KUKA KRL program: MyProgram_080().src

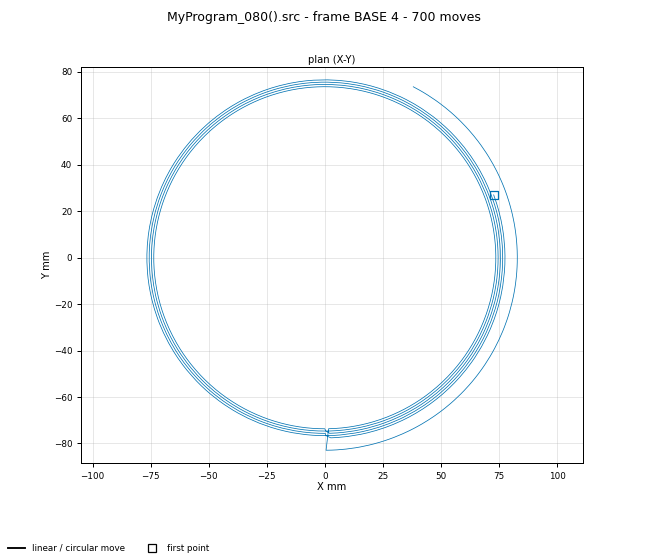
[picture p0: tool path of MyProgram_080().src in frame BASE 4, 700 of 700 moves have a stored position in this frame; points joined in program order, loops and branches not executed]
&ACCESS RVP
&REL 1
&PARAM TEMPLATE = C:\KRC\Roboter\Template\vorgabe
&PARAM EDITMASK = *
DEF MyProgram_080()
; ---- Setting reference (Base) ----
$BASE = BASE_DATA[4]

; --------------------------
; ---- Setting tool (TCP) ----
$TOOL = TOOL_DATA[3]
; --------------------------

$VEL.CP = VEL_APROX_PRINT
Startdeposition()
$VEL.CP = VEL_PRINT
LIN {X 72.7406,Y 27.0549,Z 81,A 13.4296,B 24.8995,C -2.3141,E1 25.1512,E2 431.179} C_DIS
LIN {X 74.0398,Y 23.263,Z 81,A 11.6779,B 24.8971,C -2.342,E1 25.1526,E2 432.855} C_DIS
LIN {X 75.0363,Y 19.8168,Z 81,A 8.2037,B 24.9,C -2.3088,E1 25.1553,E2 436.3875} C_DIS
LIN {X 75.8768,Y 16.3012,Z 81,A 6.032,B 24.8994,C -2.3158,E1 25.1566,E2 438.5303} C_DIS
LIN {X 76.4846,Y 13.161,Z 81,A 2.9896,B 24.9018,C -2.2877,E1 25.1581,E2 441.6211} C_DIS
LIN {X 77.0242,Y 9.5105,Z 81,A -0.3457,B 24.9041,C -2.2607,E1 25.1592,E2 445.0004} C_DIS
LIN {X 77.5014,Y 4.0671,Z 81,A -2.5659,B 24.9005,C -2.3033,E1 25.1596,E2 447.1069} C_DIS
LIN {X 77.6032,Y 0.8398,Z 81,A -5.5015,B 24.9026,C -2.2787,E1 25.1598,E2 450.0831} C_DIS
LIN {X 77.5585,Y -2.7704,Z 81,A -8.1214,B 24.9032,C -2.2716,E1 25.1596,E2 452.7042} C_DIS
LIN {X 77.3829,Y -5.9099,Z 81,A -10.3219,B 24.9035,C -2.2679,E1 25.1592,E2 454.9004} C_DIS
LIN {X 76.6451,Y -12.1903,Z 81,A -14.3809,B 24.9032,C -2.2718,E1 25.1578,E2 458.926} C_DIS
LIN {X 75.7643,Y -16.8174,Z 81,A -18.4569,B 24.9057,C -2.2423,E1 25.1557,E2 463.048} C_DIS
LIN {X 74.816,Y -20.6292,Z 81,A -21.3337,B 24.9064,C -2.2339,E1 25.1536,E2 465.928} C_DIS
LIN {X 74.0707,Y -23.163,Z 81,A -23.9313,B 24.9085,C -2.208,E1 25.1514,E2 468.5719} C_DIS
LIN {X 72.9129,Y -26.5834,Z 81,A -25.729,B 24.907,C -2.2264,E1 25.1498,E2 470.3162} C_DIS
LIN {X 71.3683,Y -30.4905,Z 81,A -29.3108,B 24.909,C -2.2023,E1 25.1459,E2 473.9352} C_DIS
LIN {X 69.9864,Y -33.5391,Z 81,A -31.3794,B 24.9086,C -2.2072,E1 25.1435,E2 475.981} C_DIS
LIN {X 67.4557,Y -38.3768,Z 81,A -35.2444,B 24.9092,C -2.2005,E1 25.1385,E2 479.8414} C_DIS
LIN {X 64.6383,Y -42.9527,Z 81,A -39.0995,B 24.9098,C -2.1927,E1 25.1328,E2 483.6954} C_DIS
LIN {X 63.2802,Y -44.929,Z 81,A -41.4223,B 24.9116,C -2.1711,E1 25.129,E2 486.0579} C_DIS
LIN {X 60.7597,Y -48.2832,Z 81,A -44.696,B 24.9127,C -2.1576,E1 25.1233,E2 489.3481} C_DIS
LIN {X 57.9727,Y -51.5963,Z 81,A -47.345,B 24.912,C -2.1659,E1 25.1185,E2 491.9656} C_DIS
LIN {X 55.8853,Y -53.8498,Z 81,A -50.1831,B 24.9139,C -2.1432,E1 25.113,E2 494.845} C_DIS
LIN {X 53.6172,Y -56.1095,Z 81,A -52.4693,B 24.9141,C -2.1399,E1 25.1084,E2 497.1295} C_DIS
LIN {X 50.5856,Y -58.8573,Z 81,A -55.0251,B 24.9136,C -2.1469,E1 25.1031,E2 499.6587} C_DIS
LIN {X 47.9048,Y -61.0588,Z 81,A -58.0995,B 24.9152,C -2.1261,E1 25.0963,E2 502.7707} C_DIS
LIN {X 45.3423,Y -62.9853,Z 81,A -59.9833,B 24.9145,C -2.1355,E1 25.0921,E2 504.6256} C_DIS
LIN {X 42.1438,Y -65.1685,Z 81,A -62.7724,B 24.9147,C -2.132,E1 25.0856,E2 507.4137} C_DIS
LIN {X 39.2698,Y -66.9396,Z 81,A -65.8722,B 24.9165,C -2.1096,E1 25.0781,E2 510.5569} C_DIS
LIN {X 36.2702,Y -68.6109,Z 81,A -67.2909,B 24.9143,C -2.138,E1 25.0748,E2 511.9043} C_DIS
LIN {X 33.3708,Y -70.0673,Z 81,A -69.9592,B 24.9152,C -2.1261,E1 25.068,E2 514.5937} C_DIS
LIN {X 29.4831,Y -71.7898,Z 81,A -73.2723,B 24.916,C -2.1164,E1 25.0595,E2 517.9219} C_DIS
LIN {X 26.0178,Y -73.117,Z 81,A -76.3261,B 24.917,C -2.1037,E1 25.0514,E2 520.9993} C_DIS
LIN {X 22.0037,Y -74.4232,Z 81,A -79.548,B 24.9175,C -2.0971,E1 25.0428,E2 524.2311} C_DIS
LIN {X 18.2814,Y -75.4238,Z 81,A -82.1856,B 24.9173,C -2.1002,E1 25.0357,E2 526.8574} C_DIS
LIN {X 15.4169,Y -76.0613,Z 81,A -84.1498,B 24.917,C -2.104,E1 25.0304,E2 528.8101} C_DIS
LIN {X 9.6899,Y -77.001,Z 81,A -88.5998,B 24.9176,C -2.0963,E1 25.0181,E2 533.2742} C_DIS
LIN {X 5.5154,Y -77.412,Z 81,A -91.4129,B 24.9171,C -2.1027,E1 25.0103,E2 536.0705} C_DIS
LIN {X 2.6067,Y -77.5643,Z 81,A -94.2953,B 24.9187,C -2.0816,E1 25.0021,E2 539.0022} C_DIS
LIN {X 2.6067,Y -77.5643,Z 81,A -94.2953,B 24.9187,C -2.0816,E1 25.0021,E2 539.0022} C_DIS
Enddeposition()
LIN {X 0.5051,Y -76.6088,Z 81,A -94.3061,B 24.914,C -2.1414,E1 25.0025,E2 538.871} C_DIS
Startdeposition()
$VEL.CP = VEL_PRINT
LIN {X 4.0039,Y -76.5168,Z 81,A -91.5176,B 24.9135,C -2.147,E1 25.0103,E2 536.0701} C_DIS
LIN {X 6.6768,Y -76.3306,Z 81,A -88.9313,B 24.9121,C -2.1645,E1 25.0176,E2 533.4436} C_DIS
LIN {X 13.1371,Y -75.4878,Z 81,A -84.5808,B 24.9131,C -2.1529,E1 25.0295,E2 529.1246} C_DIS
LIN {X 16.3512,Y -74.8562,Z 81,A -81.8311,B 24.9122,C -2.1637,E1 25.0371,E2 526.3527} C_DIS
LIN {X 19.7049,Y -74.0442,Z 81,A -79.2366,B 24.9119,C -2.1668,E1 25.0441,E2 523.755} C_DIS
LIN {X 23.4743,Y -72.9368,Z 81,A -76.6561,B 24.9125,C -2.1598,E1 25.0509,E2 521.1957} C_DIS
LIN {X 27.6858,Y -71.4453,Z 81,A -72.2914,B 24.9097,C -2.1944,E1 25.0625,E2 516.7584} C_DIS
LIN {X 31.9466,Y -69.6448,Z 81,A -69.902,B 24.9118,C -2.1679,E1 25.0684,E2 514.4377} C_DIS
LIN {X 33.9734,Y -68.6776,Z 81,A -67.9436,B 24.911,C -2.1789,E1 25.0734,E2 512.4585} C_DIS
LIN {X 38.7843,Y -66.0801,Z 81,A -64.0702,B 24.9109,C -2.1796,E1 25.0828,E2 508.5947} C_DIS
LIN {X 42.9281,Y -63.4664,Z 81,A -60.3035,B 24.9101,C -2.1898,E1 25.0917,E2 504.8164} C_DIS
LIN {X 45.9892,Y -61.2839,Z 81,A -57.4169,B 24.9094,C -2.1978,E1 25.0982,E2 501.921} C_DIS
LIN {X 49.171,Y -58.7629,Z 81,A -54.79,B 24.9099,C -2.1922,E1 25.1038,E2 499.3174} C_DIS
LIN {X 52.9625,Y -55.3703,Z 81,A -50.8405,B 24.9088,C -2.2053,E1 25.112,E2 495.3528} C_DIS
LIN {X 55.8207,Y -52.4867,Z 81,A -47.8961,B 24.9084,C -2.21,E1 25.1177,E2 492.4101} C_DIS
LIN {X 57.6696,Y -50.4483,Z 81,A -45.6064,B 24.9074,C -2.2222,E1 25.122,E2 490.1017} C_DIS
LIN {X 60.1141,Y -47.5089,Z 81,A -42.7917,B 24.9069,C -2.2284,E1 25.1269,E2 487.2855} C_DIS
LIN {X 63.1802,Y -43.3507,Z 81,A -39.3763,B 24.9071,C -2.2251,E1 25.1324,E2 483.8943} C_DIS
LIN {X 64.7091,Y -41.0307,Z 81,A -36.7547,B 24.9052,C -2.2476,E1 25.1365,E2 481.2326} C_DIS
LIN {X 66.493,Y -38.0722,Z 81,A -33.737,B 24.9035,C -2.2685,E1 25.1407,E2 478.1813} C_DIS
LIN {X 68.3146,Y -34.6981,Z 81,A -31.6623,B 24.9048,C -2.2523,E1 25.1433,E2 476.1557} C_DIS
LIN {X 69.6675,Y -31.8972,Z 81,A -29.3502,B 24.9043,C -2.2588,E1 25.1461,E2 473.8409} C_DIS
LIN {X 71.6458,Y -27.1604,Z 81,A -25.8048,B 24.9041,C -2.2614,E1 25.1498,E2 470.3089} C_DIS
LIN {X 73.3926,Y -22.0088,Z 81,A -20.8861,B 24.9007,C -2.3003,E1 25.1541,E2 465.326} C_DIS
LIN {X 74.2916,Y -18.7529,Z 81,A -18.9852,B 24.9017,C -2.2888,E1 25.1554,E2 463.4633} C_DIS
LIN {X 74.9344,Y -15.9924,Z 81,A -16.2071,B 24.8994,C -2.316,E1 25.157,E2 460.6372} C_DIS
LIN {X 75.589,Y -12.5348,Z 81,A -14.9013,B 24.9022,C -2.2833,E1 25.1576,E2 459.4164} C_DIS
LIN {X 76.1441,Y -8.5448,Z 81,A -11.2664,B 24.8997,C -2.312,E1 25.159,E2 455.735} C_DIS
LIN {X 76.4322,Y -5.3825,Z 81,A -8.9577,B 24.8992,C -2.3176,E1 25.1595,E2 453.4269} C_DIS
LIN {X 76.614,Y -1.0935,Z 81,A -5.0295,B 24.8964,C -2.3501,E1 25.1598,E2 449.4452} C_DIS
LIN {X 76.5801,Y 2.5132,Z 81,A -3.0751,B 24.8976,C -2.3356,E1 25.1596,E2 447.5368} C_DIS
LIN {X 76.4465,Y 5.1709,Z 81,A -0.1808,B 24.8946,C -2.37,E1 25.1591,E2 444.5783} C_DIS
LIN {X 76.0454,Y 9.3872,Z 81,A 2.5015,B 24.8951,C -2.3648,E1 25.1582,E2 441.9243} C_DIS
LIN {X 75.3914,Y 13.6729,Z 81,A 5.2733,B 24.8955,C -2.3603,E1 25.1569,E2 439.1792} C_DIS
LIN {X 74.78,Y 16.7004,Z 81,A 7.3071,B 24.8955,C -2.3589,E1 25.1558,E2 437.1606} C_DIS
LIN {X 74.058,Y 19.6555,Z 81,A 9.8384,B 24.8943,C -2.3737,E1 25.154,E2 434.609} C_DIS
LIN {X 73.1811,Y 22.7009,Z 81,A 12.5126,B 24.8928,C -2.3901,E1 25.1518,E2 431.9112} C_DIS
LIN {X 71.4621,Y 27.643,Z 81,A 16.0873,B 24.8928,C -2.3912,E1 25.1484,E2 428.354} C_DIS
LIN {X 70.1766,Y 30.7583,Z 81,A 19.1342,B 24.8906,C -2.4145,E1 25.145,E2 425.2688} C_DIS
LIN {X 68.8247,Y 33.6767,Z 81,A 21.4682,B 24.8902,C -2.4189,E1 25.1422,E2 422.9367} C_DIS
LIN {X 66.6712,Y 37.762,Z 81,A 24.2393,B 24.8912,C -2.4075,E1 25.1385,E2 420.2072} C_DIS
LIN {X 64.9518,Y 40.6456,Z 81,A 27.0598,B 24.8898,C -2.4234,E1 25.1344,E2 417.3634} C_DIS
LIN {X 62.8872,Y 43.7722,Z 81,A 30.8514,B 24.8864,C -2.4605,E1 25.1282,E2 413.5028} C_DIS
LIN {X 59.9348,Y 47.7358,Z 81,A 33.3959,B 24.8888,C -2.4344,E1 25.124,E2 411.0319} C_DIS
LIN {X 56.4841,Y 51.7721,Z 81,A 37.3342,B 24.888,C -2.4424,E1 25.1168,E2 407.0924} C_DIS
LIN {X 54.1841,Y 54.1766,Z 81,A 39.8561,B 24.8875,C -2.4487,E1 25.1118,E2 404.5664} C_DIS
LIN {X 51.7923,Y 56.4656,Z 81,A 42.128,B 24.8875,C -2.4477,E1 25.1072,E2 402.3062} C_DIS
LIN {X 48.7055,Y 59.1498,Z 81,A 45.1069,B 24.8872,C -2.4512,E1 25.1009,E2 399.3306} C_DIS
LIN {X 46.6152,Y 60.8101,Z 81,A 47.6684,B 24.8854,C -2.4714,E1 25.0952,E2 396.7308} C_DIS
LIN {X 41.6987,Y 64.2818,Z 81,A 51.863,B 24.8855,C -2.4697,E1 25.0855,E2 392.5543} C_DIS
LIN {X 38.5101,Y 66.2414,Z 81,A 54.7369,B 24.8849,C -2.476,E1 25.0786,E2 389.6745} C_DIS
LIN {X 35.0593,Y 68.13,Z 81,A 57.0933,B 24.8861,C -2.4631,E1 25.0729,E2 387.3554} C_DIS
LIN {X 32.717,Y 69.2862,Z 81,A 59.1876,B 24.8855,C -2.4695,E1 25.0676,E2 385.2515} C_DIS
LIN {X 27.6315,Y 71.4666,Z 81,A 64.03,B 24.8833,C -2.4938,E1 25.055,E2 380.3626} C_DIS
LIN {X 23.197,Y 73.0265,Z 81,A 67.0652,B 24.8843,C -2.4831,E1 25.0471,E2 377.3587} C_DIS
LIN {X 19.8161,Y 74.0146,Z 81,A 69.7453,B 24.884,C -2.4861,E1 25.0399,E2 374.6758} C_DIS
LIN {X 17.0226,Y 74.7067,Z 81,A 72.5334,B 24.8822,C -2.5051,E1 25.0322,E2 371.8465} C_DIS
LIN {X 13.6277,Y 75.3993,Z 81,A 74.4093,B 24.884,C -2.4862,E1 25.0272,E2 370.0177} C_DIS
LIN {X 10.5424,Y 75.8928,Z 81,A 76.8912,B 24.8835,C -2.4908,E1 25.0203,E2 367.527} C_DIS
LIN {X 5.9796,Y 76.3876,Z 81,A 80.7325,B 24.8825,C -2.5024,E1 25.0095,E2 363.6603} C_DIS
LIN {X 1.1387,Y 76.6132,Z 81,A 83.7746,B 24.884,C -2.4862,E1 25.0011,E2 360.6576} C_DIS
LIN {X -4.837,Y 76.4691,Z 81,A 88.3402,B 24.8839,C -2.4873,E1 24.9884,E2 356.0885} C_DIS
LIN {X -8.0265,Y 76.1996,Z 81,A 90.8059,B 24.8839,C -2.4881,E1 24.9815,E2 353.6197} C_DIS
LIN {X -11.1013,Y 75.8128,Z 81,A 93.1912,B 24.8838,C -2.4885,E1 24.9749,E2 351.2316} C_DIS
LIN {X -14.9837,Y 75.1429,Z 81,A 96.2499,B 24.8838,C -2.4891,E1 24.9665,E2 348.168} C_DIS
LIN {X -19.4527,Y 74.1117,Z 81,A 99.3472,B 24.8848,C -2.4771,E1 24.9582,E2 345.0951} C_DIS
LIN {X -22.985,Y 73.0928,Z 81,A 102.6998,B 24.8836,C -2.4899,E1 24.9491,E2 341.7062} C_DIS
LIN {X -26.3966,Y 71.9309,Z 81,A 105.7925,B 24.883,C -2.497,E1 24.941,E2 338.5905} C_DIS
LIN {X -30.2905,Y 70.3805,Z 81,A 107.9496,B 24.8858,C -2.467,E1 24.9356,E2 336.4998} C_DIS
LIN {X -34.5136,Y 68.4089,Z 81,A 111.2486,B 24.8867,C -2.4569,E1 24.9273,E2 333.2166} C_DIS
LIN {X -37.0817,Y 67.0511,Z 81,A 114.3662,B 24.8848,C -2.4775,E1 24.9195,E2 330.0411} C_DIS
LIN {X -40.0695,Y 65.3096,Z 81,A 116.3389,B 24.8867,C -2.457,E1 24.9149,E2 328.1109} C_DIS
LIN {X -42.8077,Y 63.5479,Z 81,A 118.7363,B 24.8872,C -2.4514,E1 24.9093,E2 325.719} C_DIS
LIN {X -46.5848,Y 60.8335,Z 81,A 122.3377,B 24.8876,C -2.4474,E1 24.9012,E2 322.1144} C_DIS
LIN {X -50.0446,Y 58.0221,Z 81,A 125.6479,B 24.8883,C -2.4395,E1 24.8941,E2 318.8104} C_DIS
LIN {X -53.7369,Y 54.6184,Z 81,A 129.1445,B 24.8897,C -2.4244,E1 24.8871,E2 315.3356} C_DIS
LIN {X -57.3893,Y 50.7688,Z 81,A 133.4156,B 24.8899,C -2.4221,E1 24.8789,E2 311.0512} C_DIS
LIN {X -60.4351,Y 47.1018,Z 81,A 136.9866,B 24.8907,C -2.413,E1 24.8726,E2 307.4854} C_DIS
LIN {X -63.3473,Y 43.104,Z 81,A 140.6648,B 24.8917,C -2.4025,E1 24.8667,E2 303.8143} C_DIS
LIN {X -65.1312,Y 40.3584,Z 81,A 142.8724,B 24.8928,C -2.3898,E1 24.8634,E2 301.6259} C_DIS
LIN {X -66.5326,Y 38.0034,Z 81,A 145.6655,B 24.8917,C -2.4021,E1 24.8594,E2 298.7886} C_DIS
LIN {X -68.4996,Y 34.3325,Z 81,A 148.3984,B 24.8934,C -2.3837,E1 24.856,E2 296.0852} C_DIS
LIN {X -70.2882,Y 30.5022,Z 81,A 152.0408,B 24.8932,C -2.3861,E1 24.8518,E2 292.4171} C_DIS
LIN {X -72.1333,Y 25.8416,Z 81,A 155.6738,B 24.8944,C -2.3718,E1 24.8483,E2 288.7978} C_DIS
LIN {X -73.6813,Y 21.0213,Z 81,A 158.6352,B 24.8972,C -2.3401,E1 24.8459,E2 285.895} C_DIS
LIN {X -74.47,Y 18.0288,Z 81,A 161.9607,B 24.8957,C -2.3573,E1 24.8436,E2 282.5089} C_DIS
LIN {X -75.456,Y 13.3139,Z 81,A 165.5401,B 24.8968,C -2.3454,E1 24.8417,E2 278.9368} C_DIS
LIN {X -75.994,Y 9.7835,Z 81,A 168.0798,B 24.8978,C -2.3337,E1 24.8408,E2 276.4099} C_DIS
LIN {X -76.4323,Y 5.3805,Z 81,A 171.932,B 24.8976,C -2.3365,E1 24.8399,E2 272.528} C_DIS
LIN {X -76.6084,Y 1.3996,Z 81,A 173.9908,B 24.9004,C -2.3045,E1 24.8398,E2 270.533} C_DIS
LIN {X -76.6007,Y -1.8197,Z 81,A 176.6959,B 24.9004,C -2.3041,E1 24.8398,E2 267.8127} C_DIS
LIN {X -76.3769,Y -6.1134,Z 81,A 179.7575,B 24.9016,C -2.2902,E1 24.8404,E2 264.7659} C_DIS
LIN {X -76.1095,Y -8.8402,Z 81,A -178.3528,B 24.9025,C -2.2799,E1 24.841,E2 262.8894} C_DIS
LIN {X -75.6777,Y -11.9906,Z 81,A -175.8658,B 24.9029,C -2.2752,E1 24.842,E2 260.399} C_DIS
LIN {X -75.009,Y -15.6367,Z 81,A -172.9725,B 24.9034,C -2.2696,E1 24.8436,E2 257.5019} C_DIS
LIN {X -74.4931,Y -17.9342,Z 81,A -170.2891,B 24.9019,C -2.2869,E1 24.8454,E2 254.7614} C_DIS
LIN {X -73.3805,Y -22.0494,Z 81,A -168.4859,B 24.9056,C -2.2434,E1 24.8467,E2 253.0518} C_DIS
LIN {X -72.0133,Y -26.1704,Z 81,A -164.7612,B 24.9054,C -2.2454,E1 24.8501,E2 249.3009} C_DIS
LIN {X -71.2631,Y -28.1496,Z 81,A -162.1753,B 24.9037,C -2.2658,E1 24.8528,E2 246.6519} C_DIS
LIN {X -69.5373,Y -32.1776,Z 81,A -159.9047,B 24.9066,C -2.2315,E1 24.8554,E2 244.4507} C_DIS
LIN {X -67.2711,Y -36.6801,Z 81,A -155.6898,B 24.9066,C -2.2323,E1 24.8608,E2 240.2115} C_DIS
LIN {X -65.0604,Y -40.4719,Z 81,A -152.7829,B 24.908,C -2.2144,E1 24.865,E2 237.3324} C_DIS
LIN {X -63.2183,Y -43.2936,Z 81,A -149.4449,B 24.9068,C -2.2287,E1 24.8703,E2 233.9437} C_DIS
LIN {X -60.9614,Y -46.4188,Z 81,A -147.5845,B 24.9096,C -2.1958,E1 24.8733,E2 232.1526} C_DIS
LIN {X -59.3245,Y -48.4924,Z 81,A -144.8184,B 24.9083,C -2.2112,E1 24.8782,E2 229.3369} C_DIS
LIN {X -55.4047,Y -52.9267,Z 81,A -140.8853,B 24.9101,C -2.1889,E1 24.8855,E2 225.4397} C_DIS
LIN {X -53.325,Y -55.0208,Z 81,A -138.8378,B 24.9108,C -2.1803,E1 24.8896,E2 223.4041} C_DIS
LIN {X -51.2072,Y -56.9969,Z 81,A -136.5265,B 24.9108,C -2.1797,E1 24.8944,E2 221.0849} C_DIS
LIN {X -49.3438,Y -58.6179,Z 81,A -134.3506,B 24.9105,C -2.1847,E1 24.899,E2 218.8886} C_DIS
LIN {X -45.6253,Y -61.555,Z 81,A -130.9776,B 24.9113,C -2.1741,E1 24.9065,E2 215.5287} C_DIS
LIN {X -43.143,Y -63.3209,Z 81,A -127.855,B 24.9098,C -2.1926,E1 24.9138,E2 212.3516} C_DIS
LIN {X -39.5137,Y -65.6474,Z 81,A -125.4562,B 24.912,C -2.166,E1 24.9194,E2 210.0085} C_DIS
LIN {X -37.3266,Y -66.9143,Z 81,A -123.4615,B 24.912,C -2.1662,E1 24.9243,E2 208.0076} C_DIS
LIN {X -33.0427,Y -69.1304,Z 81,A -119.5685,B 24.9117,C -2.1695,E1 24.9341,E2 204.0965} C_DIS
LIN {X -28.1562,Y -71.2605,Z 81,A -115.906,B 24.9128,C -2.1567,E1 24.9434,E2 200.4561} C_DIS
LIN {X -23.2066,Y -73.0234,Z 81,A -112.0862,B 24.9133,C -2.1506,E1 24.9535,E2 196.6437} C_DIS
LIN {X -20.0867,Y -73.9415,Z 81,A -108.9851,B 24.9119,C -2.1673,E1 24.962,E2 193.4979} C_DIS
LIN {X -16.5756,Y -74.8072,Z 81,A -107.0751,B 24.9138,C -2.1442,E1 24.967,E2 191.6403} C_DIS
LIN {X -13.7391,Y -75.3795,Z 81,A -104.6203,B 24.9132,C -2.1514,E1 24.9738,E2 189.1658} C_DIS
LIN {X -8.4181,Y -76.1586,Z 81,A -100.772,B 24.9136,C -2.1458,E1 24.9845,E2 185.3279} C_DIS
LIN {X -5.3144,Y -76.4368,Z 81,A -98.4403,B 24.9136,C -2.1458,E1 24.9909,E2 182.9952} C_DIS
LIN {X -2.5364,Y -76.5794,Z 81,A -96.1753,B 24.9132,C -2.1512,E1 24.9973,E2 180.7169} C_DIS
LIN {X 0.5051,Y -76.6088,Z 81,A -94.3042,B 24.9141,C -2.1406,E1 25.0025,E2 178.871} C_DIS
Enddeposition()
LIN {X 0.5051,Y -76.6088,Z 81,A -94.3042,B 24.9141,C -2.1406,E1 25.0025,E2 178.871} C_DIS
Startdeposition()
$VEL.CP = VEL_PRINT
LIN {X 0.187,Y -75.6349,Z 81,A -95.6395,B 24.9151,C -2.1275,E1 24.9987,E2 180.2374} C_DIS
LIN {X -2.5715,Y -75.5913,Z 81,A -97.6245,B 24.9149,C -2.13,E1 24.9931,E2 182.2167} C_DIS
LIN {X -5.8708,Y -75.4066,Z 81,A -100.1192,B 24.9149,C -2.1302,E1 24.9862,E2 184.7118} C_DIS
LIN {X -9.2028,Y -75.0737,Z 81,A -102.8673,B 24.9153,C -2.1249,E1 24.9785,E2 187.4742} C_DIS
LIN {X -13.0154,Y -74.5073,Z 81,A -105.9446,B 24.9156,C -2.1216,E1 24.97,E2 190.5623} C_DIS
LIN {X -18.302,Y -73.387,Z 81,A -109.9303,B 24.9152,C -2.1264,E1 24.9592,E2 194.5417} C_DIS
LIN {X -22.0543,Y -72.3487,Z 81,A -113.4366,B 24.9162,C -2.1141,E1 24.9497,E2 198.0832} C_DIS
LIN {X -25.7288,Y -71.1243,Z 81,A -115.3729,B 24.9139,C -2.1423,E1 24.9448,E2 199.9563} C_DIS
LIN {X -27.5592,Y -70.435,Z 81,A -116.8622,B 24.9139,C -2.1434,E1 24.9409,E2 201.4459} C_DIS
LIN {X -30.1071,Y -69.3842,Z 81,A -119.1075,B 24.9139,C -2.1415,E1 24.9351,E2 203.701} C_DIS
LIN {X -34.9652,Y -67.068,Z 81,A -123.3011,B 24.9139,C -2.1434,E1 24.9245,E2 207.9011} C_DIS
LIN {X -37.1553,Y -65.8801,Z 81,A -125.6886,B 24.9146,C -2.1334,E1 24.9187,E2 210.3194} C_DIS
LIN {X -41.3528,Y -63.3297,Z 81,A -128.8759,B 24.9131,C -2.1523,E1 24.9112,E2 213.4716} C_DIS
LIN {X -44.0914,Y -61.4539,Z 81,A -131.6563,B 24.9133,C -2.1498,E1 24.9048,E2 216.2676} C_DIS
LIN {X -47.6259,Y -58.7568,Z 81,A -134.8662,B 24.9125,C -2.1598,E1 24.8978,E2 219.4656} C_DIS
LIN {X -49.7101,Y -57.0044,Z 81,A -137.1254,B 24.9125,C -2.1589,E1 24.893,E2 221.7357} C_DIS
LIN {X -52.4639,Y -54.4806,Z 81,A -139.5912,B 24.9114,C -2.1735,E1 24.888,E2 224.1768} C_DIS
LIN {X -54.6745,Y -52.2627,Z 81,A -142.2119,B 24.9114,C -2.1725,E1 24.8829,E2 226.8112} C_DIS
LIN {X -57.7484,Y -48.8445,Z 81,A -145.9736,B 24.9114,C -2.1735,E1 24.876,E2 230.5874} C_DIS
LIN {X -60.5867,Y -45.2756,Z 81,A -149.6907,B 24.9112,C -2.1755,E1 24.8697,E2 234.3174} C_DIS
LIN {X -62.5842,Y -42.4714,Z 81,A -151.5252,B 24.9092,C -2.2006,E1 24.8668,E2 236.1013} C_DIS
LIN {X -64.194,Y -39.9966,Z 81,A -153.8992,B 24.909,C -2.203,E1 24.8633,E2 238.4815} C_DIS
LIN {X -66.1843,Y -36.6104,Z 81,A -157.7654,B 24.9101,C -2.1898,E1 24.8579,E2 242.3995} C_DIS
LIN {X -68.0416,Y -33.0307,Z 81,A -159.8395,B 24.9074,C -2.2213,E1 24.8554,E2 244.4094} C_DIS
LIN {X -69.7313,Y -29.2942,Z 81,A -162.8634,B 24.9065,C -2.2321,E1 24.852,E2 247.4244} C_DIS
LIN {X -70.6838,Y -26.915,Z 81,A -165.0025,B 24.9065,C -2.233,E1 24.8498,E2 249.5733} C_DIS
LIN {X -71.8569,Y -23.6037,Z 81,A -167.5533,B 24.9056,C -2.2434,E1 24.8475,E2 252.1137} C_DIS
LIN {X -72.9184,Y -20.0881,Z 81,A -170.9476,B 24.9061,C -2.2373,E1 24.8448,E2 255.5422} C_DIS
LIN {X -73.8318,Y -16.418,Z 81,A -173.6281,B 24.905,C -2.2504,E1 24.8431,E2 258.2073} C_DIS
LIN {X -74.6235,Y -12.3267,Z 81,A -176.6868,B 24.904,C -2.2624,E1 24.8416,E2 261.2553} C_DIS
LIN {X -75.0837,Y -9.118,Z 81,A -178.7345,B 24.9025,C -2.2796,E1 24.8409,E2 263.2741} C_DIS
LIN {X -75.3171,Y -6.9229,Z 81,A 178.8063,B 24.9036,C -2.2665,E1 24.8402,E2 265.7793} C_DIS
LIN {X -75.6176,Y -1.6214,Z 81,A 174.9882,B 24.9021,C -2.284,E1 24.8398,E2 269.5787} C_DIS
LIN {X -75.601,Y 2.256,Z 81,A 171.8276,B 24.9018,C -2.2882,E1 24.84,E2 272.7483} C_DIS
LIN {X -75.443,Y 5.3871,Z 81,A 169.3505,B 24.9013,C -2.2934,E1 24.8405,E2 275.2279} C_DIS
LIN {X -75.0703,Y 9.2308,Z 81,A 167.1578,B 24.899,C -2.3196,E1 24.8411,E2 277.371} C_DIS
LIN {X -74.2478,Y 14.4175,Z 81,A 162.4756,B 24.8994,C -2.3159,E1 24.8433,E2 282.09} C_DIS
LIN {X -72.9879,Y 19.8337,Z 81,A 158.8987,B 24.8969,C -2.3439,E1 24.8457,E2 285.621} C_DIS
LIN {X -71.5409,Y 24.5489,Z 81,A 154.8413,B 24.8966,C -2.3479,E1 24.8491,E2 289.6921} C_DIS
LIN {X -70.4265,Y 27.581,Z 81,A 152.4783,B 24.8957,C -2.3573,E1 24.8514,E2 292.0459} C_DIS
LIN {X -69.1035,Y 30.7478,Z 81,A 149.0769,B 24.8967,C -2.3465,E1 24.8553,E2 295.4919} C_DIS
LIN {X -67.5406,Y 34.0445,Z 81,A 147.1983,B 24.8941,C -2.3752,E1 24.8575,E2 297.3121} C_DIS
LIN {X -66.012,Y 36.919,Z 81,A 144.6887,B 24.8936,C -2.3813,E1 24.8609,E2 299.8203} C_DIS
LIN {X -64.7879,Y 39.0284,Z 81,A 142.7288,B 24.8934,C -2.3839,E1 24.8636,E2 301.7842} C_DIS
LIN {X -63.2736,Y 41.4378,Z 81,A 140.4833,B 24.893,C -2.3878,E1 24.867,E2 304.0318} C_DIS
LIN {X -60.9528,Y 44.7813,Z 81,A 137.0175,B 24.893,C -2.3871,E1 24.8727,E2 307.5161} C_DIS
LIN {X -58.3478,Y 48.1269,Z 81,A 134.1916,B 24.8915,C -2.4046,E1 24.8776,E2 310.3135} C_DIS
LIN {X -56.2904,Y 50.5172,Z 81,A 131.273,B 24.8921,C -2.398,E1 24.883,E2 313.2608} C_DIS
LIN {X -52.5398,Y 54.4074,Z 81,A 128.0897,B 24.8892,C -2.4296,E1 24.8892,E2 316.3823} C_DIS
LIN {X -51.1318,Y 55.7326,Z 81,A 126.1668,B 24.8899,C -2.422,E1 24.8931,E2 318.3314} C_DIS
LIN {X -48.6941,Y 57.8764,Z 81,A 123.1839,B 24.8906,C -2.4148,E1 24.8995,E2 321.3428} C_DIS
LIN {X -44.6967,Y 61.0147,Z 81,A 120.1082,B 24.8881,C -2.4416,E1 24.9062,E2 324.3659} C_DIS
LIN {X -42.676,Y 62.4456,Z 81,A 117.9603,B 24.8884,C -2.4386,E1 24.9112,E2 326.5282} C_DIS
LIN {X -39.9394,Y 64.2298,Z 81,A 115.4813,B 24.888,C -2.4432,E1 24.917,E2 329.0043} C_DIS
LIN {X -36.4124,Y 66.2938,Z 81,A 112.4028,B 24.8874,C -2.449,E1 24.9245,E2 332.078} C_DIS
LIN {X -34.3184,Y 67.4007,Z 81,A 109.683,B 24.8893,C -2.4292,E1 24.9314,E2 334.8522} C_DIS
LIN {X -30.6014,Y 69.1687,Z 81,A 107.7201,B 24.8862,C -2.4623,E1 24.9362,E2 336.741} C_DIS
LIN {X -27.8975,Y 70.3021,Z 81,A 105.4503,B 24.886,C -2.4642,E1 24.9421,E2 339.0115} C_DIS
LIN {X -25.5422,Y 71.1923,Z 81,A 102.5417,B 24.8881,C -2.4416,E1 24.9499,E2 341.9797} C_DIS
LIN {X -22.0661,Y 72.3437,Z 81,A 100.3654,B 24.8864,C -2.4597,E1 24.9556,E2 344.1168} C_DIS
LIN {X -19.706,Y 73.0224,Z 81,A 98.204,B 24.887,C -2.454,E1 24.9614,E2 346.2951} C_DIS
LIN {X -14.3145,Y 74.2677,Z 81,A 94.6864,B 24.885,C -2.4748,E1 24.9709,E2 349.7675} C_DIS
LIN {X -12.3246,Y 74.6238,Z 81,A 92.6064,B 24.8863,C -2.4618,E1 24.9767,E2 351.8804} C_DIS
LIN {X -8.8474,Y 75.1154,Z 81,A 90.3898,B 24.885,C -2.4748,E1 24.9828,E2 354.0676} C_DIS
LIN {X -5.8738,Y 75.4063,Z 81,A 88.1254,B 24.885,C -2.4759,E1 24.9891,E2 356.3307} C_DIS
LIN {X -1.4071,Y 75.6215,Z 81,A 84.8449,B 24.8846,C -2.4798,E1 24.9982,E2 359.6025} C_DIS
LIN {X 1.1922,Y 75.6255,Z 81,A 82.6941,B 24.885,C -2.4753,E1 25.0042,E2 361.7637} C_DIS
LIN {X 6.7431,Y 75.3337,Z 81,A 78.3874,B 24.8852,C -2.4728,E1 25.0163,E2 366.0747} C_DIS
LIN {X 9.6461,Y 75.017,Z 81,A 75.7865,B 24.8862,C -2.462,E1 25.0235,E2 368.6991} C_DIS
LIN {X 13.9063,Y 74.3461,Z 81,A 72.8857,B 24.8854,C -2.4707,E1 25.0314,E2 371.5765} C_DIS
LIN {X 17.3535,Y 73.6177,Z 81,A 70.2754,B 24.8854,C -2.4709,E1 25.0385,E2 374.1827} C_DIS
LIN {X 22.7191,Y 72.1425,Z 81,A 66.1395,B 24.8854,C -2.4702,E1 25.0496,E2 378.3133} C_DIS
LIN {X 25.0852,Y 71.3535,Z 81,A 64.1529,B 24.8859,C -2.4659,E1 25.0549,E2 380.3061} C_DIS
LIN {X 28.1192,Y 70.2145,Z 81,A 60.933,B 24.888,C -2.4426,E1 25.0634,E2 383.574} C_DIS
LIN {X 31.6269,Y 68.7054,Z 81,A 59.1843,B 24.8854,C -2.4708,E1 25.0677,E2 385.2516} C_DIS
LIN {X 33.8533,Y 67.636,Z 81,A 57.2317,B 24.8858,C -2.4663,E1 25.0726,E2 387.2097} C_DIS
LIN {X 37.0704,Y 65.9274,Z 81,A 53.7248,B 24.8881,C -2.4418,E1 25.0813,E2 390.7646} C_DIS
LIN {X 41.0337,Y 63.5364,Z 81,A 50.5662,B 24.8877,C -2.4462,E1 25.0887,E2 393.9027} C_DIS
LIN {X 44.5353,Y 61.1329,Z 81,A 47.2813,B 24.8884,C -2.4389,E1 25.0962,E2 397.1934} C_DIS
LIN {X 47.6073,Y 58.7719,Z 81,A 44.406,B 24.8887,C -2.4353,E1 25.1025,E2 400.0666} C_DIS
LIN {X 50.3754,Y 56.4174,Z 81,A 41.8904,B 24.8886,C -2.4367,E1 25.1078,E2 402.5689} C_DIS
LIN {X 52.7262,Y 54.2278,Z 81,A 39.4359,B 24.8891,C -2.4311,E1 25.1127,E2 405.0266} C_DIS
LIN {X 54.9304,Y 51.9933,Z 81,A 37.0876,B 24.8895,C -2.4268,E1 25.1173,E2 407.3748} C_DIS
LIN {X 57.9406,Y 48.617,Z 81,A 33.6958,B 24.8901,C -2.4201,E1 25.1235,E2 410.7672} C_DIS
LIN {X 60.7715,Y 45.0289,Z 81,A 29.605,B 24.8925,C -2.3936,E1 25.1305,E2 414.9013} C_DIS
LIN {X 62.661,Y 42.3579,Z 81,A 26.6602,B 24.8942,C -2.374,E1 25.1352,E2 417.8779} C_DIS
LIN {X 65.162,Y 38.3994,Z 81,A 24.2775,B 24.892,C -2.3985,E1 25.1385,E2 420.1905} C_DIS
LIN {X 66.6855,Y 35.6905,Z 81,A 21.7547,B 24.8931,C -2.3872,E1 25.1419,E2 422.7268} C_DIS
LIN {X 67.8393,Y 33.4431,Z 81,A 19.6052,B 24.8942,C -2.375,E1 25.1446,E2 424.8937} C_DIS
LIN {X 69.9497,Y 28.7698,Z 81,A 16.4931,B 24.8931,C -2.3868,E1 25.148,E2 427.9609} C_DIS
LIN {X 71.4411,Y 24.8356,Z 81,A 12.5801,B 24.8958,C -2.356,E1 25.1518,E2 431.9247} C_DIS
LIN {X 72.6249,Y 21.1276,Z 81,A 9.9842,B 24.8958,C -2.3576,E1 25.1539,E2 434.502} C_DIS
LIN {X 73.5552,Y 17.6161,Z 81,A 7.2599,B 24.8964,C -2.3501,E1 25.1558,E2 437.2283} C_DIS
LIN {X 74.2544,Y 14.3835,Z 81,A 4.8353,B 24.8968,C -2.3448,E1 25.1572,E2 439.6513} C_DIS
LIN {X 74.7771,Y 11.3584,Z 81,A 2.3403,B 24.8979,C -2.3325,E1 25.1583,E2 442.1606} C_DIS
LIN {X 75.3727,Y 6.2945,Z 81,A -1.2968,B 24.8984,C -2.3271,E1 25.1594,E2 445.789} C_DIS
LIN {X 75.5687,Y 3.1576,Z 81,A -3.7317,B 24.8992,C -2.318,E1 25.1597,E2 448.231} C_DIS
LIN {X 75.6284,Y -1.0305,Z 81,A -6.9286,B 24.9001,C -2.3072,E1 25.1597,E2 451.4345} C_DIS
LIN {X 75.5444,Y -3.7184,Z 81,A -8.8511,B 24.9004,C -2.3041,E1 25.1595,E2 453.3527} C_DIS
LIN {X 75.351,Y -6.5559,Z 81,A -10.982,B 24.9009,C -2.2979,E1 25.159,E2 455.4856} C_DIS
LIN {X 75.0263,Y -9.5742,Z 81,A -13.6675,B 24.9026,C -2.2791,E1 25.1581,E2 458.1997} C_DIS
LIN {X 74.5384,Y -12.8359,Z 81,A -16.0757,B 24.903,C -2.2738,E1 25.157,E2 460.6062} C_DIS
LIN {X 73.9105,Y -16.0572,Z 81,A -18.1471,B 24.9026,C -2.2784,E1 25.1559,E2 462.6548} C_DIS
LIN {X 73.2293,Y -18.9227,Z 81,A -20.7508,B 24.9042,C -2.2602,E1 25.1541,E2 465.2863} C_DIS
LIN {X 71.9087,Y -23.447,Z 81,A -24.4536,B 24.9054,C -2.2452,E1 25.151,E2 469.0035} C_DIS
LIN {X 70.867,Y -26.4311,Z 81,A -26.7938,B 24.9059,C -2.2394,E1 25.1488,E2 471.3443} C_DIS
LIN {X 69.2502,Y -30.4146,Z 81,A -29.5515,B 24.9055,C -2.2445,E1 25.1458,E2 474.0748} C_DIS
LIN {X 67.9561,Y -33.2077,Z 81,A -31.9138,B 24.9062,C -2.2366,E1 25.1429,E2 476.443} C_DIS
LIN {X 66.0662,Y -36.8219,Z 81,A -35.192,B 24.9074,C -2.2221,E1 25.1386,E2 479.7384} C_DIS
LIN {X 63.3488,Y -41.3238,Z 81,A -38.9177,B 24.9077,C -2.2185,E1 25.1331,E2 483.4538} C_DIS
LIN {X 61.2511,Y -44.372,Z 81,A -41.7265,B 24.9083,C -2.2106,E1 25.1286,E2 486.2672} C_DIS
LIN {X 59.4685,Y -46.7346,Z 81,A -44.1847,B 24.9094,C -2.1983,E1 25.1244,E2 488.743} C_DIS
LIN {X 56.5204,Y -50.2603,Z 81,A -47.3637,B 24.9094,C -2.1983,E1 25.1186,E2 491.9076} C_DIS
LIN {X 53.7801,Y -53.1817,Z 81,A -50.6248,B 24.9105,C -2.1842,E1 25.1123,E2 495.188} C_DIS
LIN {X 50.8711,Y -55.9698,Z 81,A -53.8387,B 24.9115,C -2.1724,E1 25.1057,E2 498.4166} C_DIS
LIN {X 48.0019,Y -58.4517,Z 81,A -56.8346,B 24.9123,C -2.1624,E1 25.0993,E2 501.4245} C_DIS
LIN {X 44.1259,Y -61.4293,Z 81,A -60.3026,B 24.9123,C -2.1615,E1 25.0915,E2 504.8823} C_DIS
LIN {X 41.2801,Y -63.3776,Z 81,A -62.4035,B 24.9116,C -2.1712,E1 25.0867,E2 506.9533} C_DIS
LIN {X 39.3089,Y -64.6173,Z 81,A -65.1713,B 24.9142,C -2.1392,E1 25.0799,E2 509.7881} C_DIS
LIN {X 36.0647,Y -66.4825,Z 81,A -67.3438,B 24.9131,C -2.1531,E1 25.0747,E2 511.9215} C_DIS
LIN {X 32.8711,Y -68.1183,Z 81,A -69.8606,B 24.9129,C -2.1544,E1 25.0685,E2 514.4284} C_DIS
LIN {X 28.8442,Y -69.9185,Z 81,A -73.2307,B 24.9134,C -2.1486,E1 25.0598,E2 517.804} C_DIS
LIN {X 25.4581,Y -71.2218,Z 81,A -75.9738,B 24.9137,C -2.1451,E1 25.0526,E2 520.5495} C_DIS
LIN {X 23.0078,Y -72.0508,Z 81,A -78.0833,B 24.9142,C -2.1385,E1 25.047,E2 522.6706} C_DIS
LIN {X 18.3991,Y -73.3639,Z 81,A -81.6616,B 24.9144,C -2.1361,E1 25.0374,E2 526.2489} C_DIS
LIN {X 15.5847,Y -74.0125,Z 81,A -83.7835,B 24.9144,C -2.136,E1 25.0316,E2 528.3683} C_DIS
LIN {X 12.4935,Y -74.5956,Z 81,A -86.3693,B 24.915,C -2.1286,E1 25.0244,E2 530.9689} C_DIS
LIN {X 7.8478,Y -75.2264,Z 81,A -89.5063,B 24.9143,C -2.1377,E1 25.0158,E2 534.0817} C_DIS
LIN {X 5.2508,Y -75.4523,Z 81,A -91.6189,B 24.9147,C -2.133,E1 25.0099,E2 536.2044} C_DIS
LIN {X 2.0909,Y -75.606,Z 81,A -94.1727,B 24.9151,C -2.1279,E1 25.0027,E2 538.7697} C_DIS
LIN {X 2.0909,Y -75.606,Z 81,A -94.1727,B 24.9151,C -2.1279,E1 25.0027,E2 538.7697} C_DIS
Enddeposition()
LIN {X 0.4909,Y -74.6447,Z 81,A -95.1334,B 24.9132,C -2.1517,E1 25.0002,E2 539.6738} C_DIS
Startdeposition()
$VEL.CP = VEL_PRINT
LIN {X 2.4368,Y -74.6084,Z 81,A -92.7552,B 24.9112,C -2.176,E1 25.007,E2 537.2383} C_DIS
LIN {X 5.3562,Y -74.4563,Z 81,A -90.4446,B 24.911,C -2.1788,E1 25.0135,E2 534.9221} C_DIS
LIN {X 8.4096,Y -74.1733,Z 81,A -88.0612,B 24.9108,C -2.1809,E1 25.0201,E2 532.5352} C_DIS
LIN {X 11.8495,Y -73.7029,Z 81,A -85.409,B 24.9107,C -2.1824,E1 25.0274,E2 529.8818} C_DIS
LIN {X 14.9272,Y -73.1404,Z 81,A -83.0928,B 24.9107,C -2.1821,E1 25.0338,E2 527.5692} C_DIS
LIN {X 17.9019,Y -72.4699,Z 81,A -80.3653,B 24.9096,C -2.1952,E1 25.0412,E2 524.8145} C_DIS
LIN {X 22.7431,Y -71.0995,Z 81,A -77.2322,B 24.9109,C -2.179,E1 25.0495,E2 521.7252} C_DIS
LIN {X 25.3826,Y -70.2004,Z 81,A -74.5797,B 24.9095,C -2.1962,E1 25.0566,E2 519.0373} C_DIS
LIN {X 28.4637,Y -69.0092,Z 81,A -72.1579,B 24.9095,C -2.1965,E1 25.0629,E2 516.6203} C_DIS
LIN {X 31.2836,Y -67.777,Z 81,A -70.1135,B 24.91,C -2.191,E1 25.068,E2 514.594} C_DIS
LIN {X 33.2772,Y -66.8204,Z 81,A -68.1889,B 24.9092,C -2.2002,E1 25.0729,E2 512.6526} C_DIS
LIN {X 35.9616,Y -65.4161,Z 81,A -65.6746,B 24.9084,C -2.2096,E1 25.0791,E2 510.1233} C_DIS
LIN {X 39.1979,Y -63.5297,Z 81,A -62.9158,B 24.9083,C -2.2115,E1 25.0857,E2 507.3685} C_DIS
LIN {X 41.8996,Y -61.7798,Z 81,A -60.4959,B 24.908,C -2.2149,E1 25.0913,E2 504.9487} C_DIS
LIN {X 44.8023,Y -59.7083,Z 81,A -57.0245,B 24.9057,C -2.2421,E1 25.0993,E2 501.4253} C_DIS
LIN {X 47.6739,Y -57.4415,Z 81,A -55.5094,B 24.9084,C -2.2103,E1 25.1024,E2 499.9912} C_DIS
LIN {X 50.0298,Y -55.4009,Z 81,A -52.3874,B 24.9061,C -2.2371,E1 25.109,E2 496.8182} C_DIS
LIN {X 53.3822,Y -52.1788,Z 81,A -48.6023,B 24.9049,C -2.252,E1 25.1165,E2 493.0137} C_DIS
LIN {X 57.1611,Y -48.0098,Z 81,A -44.5307,B 24.9046,C -2.2556,E1 25.124,E2 488.9519} C_DIS
LIN {X 59.5231,Y -45.0488,Z 81,A -41.3006,B 24.9031,C -2.273,E1 25.1296,E2 485.696} C_DIS
LIN {X 61.6544,Y -42.0849,Z 81,A -39.1361,B 24.904,C -2.2616,E1 25.133,E2 483.5691} C_DIS
LIN {X 63.2125,Y -39.7056,Z 81,A -36.9222,B 24.9034,C -2.2686,E1 25.1363,E2 481.3497} C_DIS
LIN {X 65.6349,Y -35.5583,Z 81,A -33.3996,B 24.903,C -2.2743,E1 25.1412,E2 477.8318} C_DIS
LIN {X 66.881,Y -33.155,Z 81,A -31.2496,B 24.9023,C -2.2826,E1 25.1439,E2 475.6738} C_DIS
LIN {X 68.2571,Y -30.2238,Z 81,A -28.6148,B 24.9012,C -2.2945,E1 25.147,E2 473.0253} C_DIS
LIN {X 69.6223,Y -26.9279,Z 81,A -26.271,B 24.9015,C -2.291,E1 25.1494,E2 470.7027} C_DIS
LIN {X 70.3541,Y -24.9538,Z 81,A -24.101,B 24.8997,C -2.3126,E1 25.1515,E2 468.4938} C_DIS
LIN {X 71.7906,Y -20.4558,Z 81,A -20.8763,B 24.8997,C -2.3118,E1 25.1541,E2 465.2893} C_DIS
LIN {X 72.555,Y -17.5533,Z 81,A -18.577,B 24.8991,C -2.3189,E1 25.1557,E2 462.9865} C_DIS
LIN {X 73.1983,Y -14.6449,Z 81,A -16.13,B 24.8981,C -2.331,E1 25.1571,E2 460.5253} C_DIS
LIN {X 73.8314,Y -11.0185,Z 81,A -13.6615,B 24.8982,C -2.3292,E1 25.1582,E2 458.0756} C_DIS
LIN {X 74.1296,Y -8.783,Z 81,A -11.7866,B 24.8973,C -2.339,E1 25.1588,E2 456.1884} C_DIS
LIN {X 74.4431,Y -5.5421,Z 81,A -9.2157,B 24.8965,C -2.3491,E1 25.1595,E2 453.6089} C_DIS
LIN {X 74.603,Y -2.6111,Z 81,A -6.9702,B 24.8958,C -2.3561,E1 25.1597,E2 451.3603} C_DIS
LIN {X 74.6484,Y 0.1829,Z 81,A -4.9094,B 24.8955,C -2.3604,E1 25.1597,E2 449.3016} C_DIS
LIN {X 74.5908,Y 2.9354,Z 81,A -2.8117,B 24.8949,C -2.3666,E1 25.1596,E2 447.2017} C_DIS
LIN {X 74.4303,Y 5.7027,Z 81,A -0.7107,B 24.8944,C -2.3726,E1 25.1592,E2 445.099} C_DIS
LIN {X 74.1251,Y 8.8211,Z 81,A 1.4148,B 24.8944,C -2.3717,E1 25.1586,E2 442.9881} C_DIS
LIN {X 73.8234,Y 11.0698,Z 81,A 3.4954,B 24.893,C -2.3873,E1 25.1577,E2 440.8829} C_DIS
LIN {X 73.2992,Y 14.1265,Z 81,A 5.8653,B 24.8924,C -2.3944,E1 25.1566,E2 438.5103} C_DIS
LIN {X 72.6489,Y 17.1641,Z 81,A 8.2457,B 24.8918,C -2.4015,E1 25.1551,E2 436.1268} C_DIS
LIN {X 71.8229,Y 20.3419,Z 81,A 10.6979,B 24.8913,C -2.4071,E1 25.1533,E2 433.6754} C_DIS
LIN {X 70.0668,Y 25.7487,Z 81,A 14.7886,B 24.8908,C -2.4118,E1 25.1497,E2 429.5968} C_DIS
LIN {X 69.2355,Y 27.9075,Z 81,A 16.8309,B 24.8897,C -2.4248,E1 25.1476,E2 427.5351} C_DIS
LIN {X 66.9858,Y 32.9436,Z 81,A 20.8723,B 24.8891,C -2.431,E1 25.1429,E2 423.501} C_DIS
LIN {X 65.7644,Y 35.3194,Z 81,A 23.0559,B 24.8882,C -2.4405,E1 25.14,E2 421.3064} C_DIS
LIN {X 64.1988,Y 38.0901,Z 81,A 25.8658,B 24.8866,C -2.4578,E1 25.136,E2 418.4701} C_DIS
LIN {X 61.9571,Y 41.6378,Z 81,A 28.691,B 24.8869,C -2.4543,E1 25.1318,E2 415.6672} C_DIS
LIN {X 60.019,Y 44.3867,Z 81,A 31.9511,B 24.8845,C -2.4806,E1 25.1263,E2 412.3608} C_DIS
LIN {X 57.8879,Y 47.1311,Z 81,A 33.5426,B 24.8868,C -2.4555,E1 25.1237,E2 410.8361} C_DIS
LIN {X 56.3386,Y 48.9727,Z 81,A 35.7484,B 24.8855,C -2.4701,E1 25.1196,E2 408.6057} C_DIS
LIN {X 54.1346,Y 51.3994,Z 81,A 38.2717,B 24.885,C -2.4758,E1 25.1148,E2 406.0801} C_DIS
LIN {X 51.9934,Y 53.5638,Z 81,A 40.5454,B 24.8847,C -2.4789,E1 25.1103,E2 403.8086} C_DIS
LIN {X 49.6854,Y 55.7109,Z 81,A 43.032,B 24.884,C -2.4856,E1 25.1051,E2 401.3161} C_DIS
LIN {X 47.2962,Y 57.754,Z 81,A 45.3853,B 24.8838,C -2.4884,E1 25.1001,E2 398.9652} C_DIS
LIN {X 44.4993,Y 59.9338,Z 81,A 49.006,B 24.8809,C -2.519,E1 25.0919,E2 395.2852} C_DIS
LIN {X 41.1386,Y 62.2892,Z 81,A 50.9976,B 24.8835,C -2.491,E1 25.0875,E2 393.3664} C_DIS
LIN {X 39.2164,Y 63.5181,Z 81,A 52.9672,B 24.8827,C -2.4998,E1 25.0828,E2 391.3823} C_DIS
LIN {X 36.7779,Y 64.9608,Z 81,A 55.7636,B 24.8808,C -2.5204,E1 25.0759,E2 388.5454} C_DIS
LIN {X 33.9554,Y 66.4782,Z 81,A 57.6185,B 24.8821,C -2.5066,E1 25.0714,E2 386.7285} C_DIS
LIN {X 31.4452,Y 67.7017,Z 81,A 59.9308,B 24.8814,C -2.5138,E1 25.0655,E2 384.405} C_DIS
LIN {X 28.4464,Y 69.0162,Z 81,A 62.2486,B 24.8816,C -2.5111,E1 25.0596,E2 382.0992} C_DIS
LIN {X 25.5114,Y 70.1534,Z 81,A 64.5968,B 24.8816,C -2.5115,E1 25.0534,E2 379.755} C_DIS
LIN {X 22.6437,Y 71.1317,Z 81,A 67.0723,B 24.881,C -2.5174,E1 25.0468,E2 377.2702} C_DIS
LIN {X 18.5517,Y 72.306,Z 81,A 69.9846,B 24.8817,C -2.5099,E1 25.0391,E2 374.3805} C_DIS
LIN {X 14.8897,Y 73.1477,Z 81,A 73.3286,B 24.8804,C -2.5238,E1 25.0299,E2 371.008} C_DIS
LIN {X 10.9931,Y 73.8336,Z 81,A 76.3861,B 24.8803,C -2.5253,E1 25.0214,E2 367.9499} C_DIS
LIN {X 7.5142,Y 74.2693,Z 81,A 79.196,B 24.88,C -2.5288,E1 25.0136,E2 365.1334} C_DIS
LIN {X 2.5325,Y 74.6054,Z 81,A 82.2961,B 24.8818,C -2.5093,E1 25.0051,E2 362.0809} C_DIS
LIN {X -0.8928,Y 74.6439,Z 81,A 85.3289,B 24.8808,C -2.5195,E1 24.9966,E2 359.0242} C_DIS
LIN {X -4.285,Y 74.5251,Z 81,A 87.6523,B 24.8816,C -2.5112,E1 24.9901,E2 356.7199} C_DIS
LIN {X -6.7213,Y 74.3449,Z 81,A 89.7623,B 24.8811,C -2.5165,E1 24.9842,E2 354.5964} C_DIS
LIN {X -9.8929,Y 73.9902,Z 81,A 93.0331,B 24.8792,C -2.5364,E1 24.975,E2 351.2758} C_DIS
LIN {X -13.5805,Y 73.4032,Z 81,A 94.8434,B 24.882,C -2.507,E1 24.9703,E2 349.5337} C_DIS
LIN {X -17.0284,Y 72.6802,Z 81,A 98.3181,B 24.8804,C -2.5244,E1 24.9607,E2 346.0133} C_DIS
LIN {X -21.1436,Y 71.5911,Z 81,A 101.8911,B 24.88,C -2.5287,E1 24.951,E2 342.4241} C_DIS
LIN {X -24.6866,Y 70.4478,Z 81,A 103.9102,B 24.8823,C -2.5039,E1 24.9458,E2 340.4602} C_DIS
LIN {X -27.6015,Y 69.3584,Z 81,A 106.4073,B 24.8823,C -2.5035,E1 24.9393,E2 337.9588} C_DIS
LIN {X -30.5466,Y 68.112,Z 81,A 109.7009,B 24.8807,C -2.521,E1 24.9308,E2 334.6154} C_DIS
LIN {X -34.118,Y 66.3952,Z 81,A 111.6903,B 24.8836,C -2.4898,E1 24.926,E2 332.6952} C_DIS
LIN {X -36.7281,Y 64.9886,Z 81,A 113.9187,B 24.8841,C -2.4848,E1 24.9206,E2 330.4724} C_DIS
LIN {X -38.6434,Y 63.8673,Z 81,A 115.8056,B 24.884,C -2.4862,E1 24.916,E2 328.5763} C_DIS
LIN {X -41.0856,Y 62.3242,Z 81,A 118.0263,B 24.8844,C -2.4821,E1 24.9108,E2 326.3581} C_DIS
LIN {X -43.7137,Y 60.5114,Z 81,A 120.5641,B 24.8846,C -2.4794,E1 24.905,E2 323.8183} C_DIS
LIN {X -46.079,Y 58.7292,Z 81,A 122.7909,B 24.8852,C -2.4735,E1 24.9001,E2 321.5974} C_DIS
LIN {X -47.7954,Y 57.3405,Z 81,A 124.5289,B 24.8854,C -2.4709,E1 24.8964,E2 319.859} C_DIS
LIN {X -50.1964,Y 55.252,Z 81,A 127.0614,B 24.8857,C -2.4675,E1 24.8911,E2 317.3244} C_DIS
LIN {X -52.5929,Y 52.9749,Z 81,A 129.7143,B 24.886,C -2.4644,E1 24.8858,E2 314.668} C_DIS
LIN {X -55.0923,Y 50.3704,Z 81,A 132.3935,B 24.8868,C -2.4554,E1 24.8807,E2 311.9986} C_DIS
LIN {X -57.2072,Y 47.9559,Z 81,A 134.8349,B 24.8875,C -2.4486,E1 24.8762,E2 309.5623} C_DIS
LIN {X -59.3275,Y 45.3064,Z 81,A 137.5676,B 24.8878,C -2.4448,E1 24.8715,E2 306.8257} C_DIS
LIN {X -61.0868,Y 42.9052,Z 81,A 139.8247,B 24.8885,C -2.4379,E1 24.8679,E2 304.5739} C_DIS
LIN {X -62.9101,Y 40.183,Z 81,A 142.2404,B 24.8893,C -2.4286,E1 24.8642,E2 302.1682} C_DIS
LIN {X -64.4402,Y 37.6817,Z 81,A 144.5258,B 24.8898,C -2.4231,E1 24.8609,E2 299.8843} C_DIS
LIN {X -65.9251,Y 35.0182,Z 81,A 146.8482,B 24.8905,C -2.4159,E1 24.8578,E2 297.5668} C_DIS
LIN {X -67.7099,Y 31.4278,Z 81,A 149.6861,B 24.8918,C -2.4012,E1 24.8544,E2 294.7486} C_DIS
LIN {X -68.6543,Y 29.3092,Z 81,A 151.8092,B 24.8916,C -2.4039,E1 24.852,E2 292.6073} C_DIS
LIN {X -69.8541,Y 26.3201,Z 81,A 154.3224,B 24.8921,C -2.3974,E1 24.8495,E2 290.0957} C_DIS
LIN {X -70.961,Y 23.1711,Z 81,A 157.0852,B 24.8924,C -2.3943,E1 24.847,E2 287.3246} C_DIS
LIN {X -71.847,Y 20.2568,Z 81,A 159.2392,B 24.8935,C -2.3827,E1 24.8453,E2 285.1859} C_DIS
LIN {X -72.9775,Y 15.705,Z 81,A 162.8285,B 24.8945,C -2.3711,E1 24.843,E2 281.6031} C_DIS
LIN {X -73.5642,Y 12.6799,Z 81,A 165.2278,B 24.8951,C -2.3644,E1 24.8418,E2 279.2055} C_DIS
LIN {X -74.0411,Y 9.5001,Z 81,A 168.6929,B 24.8937,C -2.3801,E1 24.8406,E2 275.6822} C_DIS
LIN {X -74.4647,Y 5.2313,Z 81,A 171.0799,B 24.8965,C -2.3482,E1 24.8401,E2 273.3571} C_DIS
LIN {X -74.5976,Y 2.7766,Z 81,A 172.9667,B 24.8971,C -2.3422,E1 24.8398,E2 271.4733} C_DIS
LIN {X -74.6344,Y -1.4232,Z 81,A 176.2835,B 24.8978,C -2.3342,E1 24.8398,E2 268.1557} C_DIS
LIN {X -74.4605,Y -5.2881,Z 81,A 179.1807,B 24.8987,C -2.3231,E1 24.8403,E2 265.2675} C_DIS
LIN {X -74.2763,Y -7.4475,Z 81,A -179.1614,B 24.8992,C -2.3177,E1 24.8408,E2 263.6126} C_DIS
LIN {X -73.7278,Y -11.6881,Z 81,A -175.8021,B 24.8999,C -2.3093,E1 24.8421,E2 260.2533} C_DIS
LIN {X -72.8781,Y -16.1608,Z 81,A -172.573,B 24.9014,C -2.2923,E1 24.8438,E2 257.0456} C_DIS
LIN {X -72.2922,Y -18.6054,Z 81,A -170.4673,B 24.9016,C -2.2906,E1 24.8453,E2 254.9317} C_DIS
LIN {X -71.0228,Y -22.9802,Z 81,A -166.9636,B 24.9024,C -2.2804,E1 24.8481,E2 251.4323} C_DIS
LIN {X -70.3148,Y -25.0658,Z 81,A -165.2232,B 24.9028,C -2.2766,E1 24.8497,E2 249.6911} C_DIS
LIN {X -69.3563,Y -27.6069,Z 81,A -163.0327,B 24.9031,C -2.2731,E1 24.8519,E2 247.4966} C_DIS
LIN {X -68.1409,Y -30.4826,Z 81,A -160.6701,B 24.9037,C -2.2655,E1 24.8545,E2 245.139} C_DIS
LIN {X -66.4251,Y -34.0593,Z 81,A -157.3937,B 24.9039,C -2.2627,E1 24.8586,E2 241.8517} C_DIS
LIN {X -64.8307,Y -37.0047,Z 81,A -155.2291,B 24.9054,C -2.2461,E1 24.8615,E2 239.7154} C_DIS
LIN {X -63.5159,Y -39.22,Z 81,A -153.0283,B 24.9054,C -2.2463,E1 24.8647,E2 237.5028} C_DIS
LIN {X -61.9821,Y -41.6009,Z 81,A -150.8025,B 24.9057,C -2.2421,E1 24.8681,E2 235.276} C_DIS
LIN {X -59.4946,Y -45.0868,Z 81,A -147.5527,B 24.9064,C -2.2332,E1 24.8735,E2 232.0316} C_DIS
LIN {X -57.6127,Y -47.4679,Z 81,A -144.1985,B 24.9048,C -2.253,E1 24.8795,E2 228.6145} C_DIS
LIN {X -54.7768,Y -50.7143,Z 81,A -142.0889,B 24.9079,C -2.216,E1 24.8834,E2 226.5838} C_DIS
LIN {X -52.8184,Y -52.7514,Z 81,A -139.6709,B 24.9078,C -2.2176,E1 24.8881,E2 224.1518} C_DIS
LIN {X -50.5866,Y -54.894,Z 81,A -137.0594,B 24.9077,C -2.2187,E1 24.8934,E2 221.5268} C_DIS
LIN {X -47.6896,Y -57.4284,Z 81,A -133.2332,B 24.9063,C -2.2352,E1 24.9018,E2 217.6467} C_DIS
LIN {X -44.0547,Y -60.262,Z 81,A -131.1377,B 24.9098,C -2.1926,E1 24.9062,E2 215.6452} C_DIS
LIN {X -42.4626,Y -61.3945,Z 81,A -129.2376,B 24.9092,C -2.2002,E1 24.9106,E2 213.7205} C_DIS
LIN {X -39.7998,Y -63.1537,Z 81,A -126.8344,B 24.9096,C -2.1953,E1 24.9163,E2 211.3213} C_DIS
LIN {X -36.4395,Y -65.1498,Z 81,A -124.3395,B 24.911,C -2.1783,E1 24.9222,E2 208.8594} C_DIS
LIN {X -34.6181,Y -66.1358,Z 81,A -122.1036,B 24.9098,C -2.1927,E1 24.9278,E2 206.583} C_DIS
LIN {X -32.2013,Y -67.3456,Z 81,A -120.1564,B 24.9103,C -2.1869,E1 24.9327,E2 204.6444} C_DIS
LIN {X -29.4852,Y -68.5791,Z 81,A -117.8171,B 24.9103,C -2.1857,E1 24.9387,E2 202.3024} C_DIS
LIN {X -26.7367,Y -69.6963,Z 81,A -115.571,B 24.9106,C -2.1828,E1 24.9445,E2 200.0585} C_DIS
LIN {X -23.76,Y -70.7658,Z 81,A -113.1567,B 24.9108,C -2.1804,E1 24.9508,E2 197.6451} C_DIS
LIN {X -21.0866,Y -71.608,Z 81,A -111.1838,B 24.9113,C -2.1742,E1 24.9561,E2 195.6835} C_DIS
LIN {X -17.8679,Y -72.4782,Z 81,A -108.2588,B 24.9107,C -2.1824,E1 24.9641,E2 192.7349} C_DIS
LIN {X -14.432,Y -73.2393,Z 81,A -105.5982,B 24.9108,C -2.1801,E1 24.9713,E2 190.0763} C_DIS
LIN {X -11.4099,Y -73.7709,Z 81,A -103.4425,B 24.9113,C -2.1741,E1 24.9772,E2 187.9329} C_DIS
LIN {X -8.8724,Y -74.1191,Z 81,A -101.4409,B 24.9113,C -2.1747,E1 24.9828,E2 185.9285} C_DIS
LIN {X -5.963,Y -74.4095,Z 81,A -99.2093,B 24.9113,C -2.1743,E1 24.989,E2 183.6969} C_DIS
LIN {X -2.7374,Y -74.5991,Z 81,A -96.5615,B 24.9109,C -2.179,E1 24.9964,E2 181.0372} C_DIS
LIN {X 0.4909,Y -74.6447,Z 81,A -95.1322,B 24.9132,C -2.1512,E1 25.0002,E2 179.6738} C_DIS
Enddeposition()
LIN {X 0.4909,Y -74.6447,Z 81,A -95.1322,B 24.9132,C -2.1512,E1 25.0002,E2 179.6738} C_DIS
Startdeposition()
$VEL.CP = VEL_PRINT
LIN {X -0.0131,Y -73.6627,Z 81,A -95.7532,B 24.9123,C -2.1623,E1 24.9986,E2 180.2685} C_DIS
LIN {X -2.7185,Y -73.6126,Z 81,A -97.8017,B 24.9123,C -2.1635,E1 24.9928,E2 182.3144} C_DIS
LIN {X -5.4205,Y -73.4631,Z 81,A -99.9464,B 24.9123,C -2.1624,E1 24.9869,E2 184.4624} C_DIS
LIN {X -8.1153,Y -73.2144,Z 81,A -102.0125,B 24.9122,C -2.1636,E1 24.9811,E2 186.5269} C_DIS
LIN {X -10.8175,Y -72.8641,Z 81,A -104.1651,B 24.9122,C -2.1632,E1 24.9752,E2 188.6821} C_DIS
LIN {X -13.6755,Y -72.3813,Z 81,A -106.3622,B 24.912,C -2.1655,E1 24.9691,E2 190.8761} C_DIS
LIN {X -16.2172,Y -71.855,Z 81,A -108.3857,B 24.912,C -2.1662,E1 24.9636,E2 192.9003} C_DIS
LIN {X -18.8004,Y -71.2231,Z 81,A -110.5158,B 24.912,C -2.1658,E1 24.9578,E2 195.0344} C_DIS
LIN {X -21.789,Y -70.3651,Z 81,A -112.8427,B 24.9117,C -2.1698,E1 24.9516,E2 197.3557} C_DIS
LIN {X -24.4636,Y -69.4805,Z 81,A -114.9898,B 24.9115,C -2.1727,E1 24.9459,E2 199.5} C_DIS
LIN {X -26.8847,Y -68.58,Z 81,A -117.0481,B 24.9115,C -2.1733,E1 24.9406,E2 201.5611} C_DIS
LIN {X -29.4904,Y -67.5006,Z 81,A -119.3989,B 24.9115,C -2.1717,E1 24.9345,E2 203.9213} C_DIS
LIN {X -32.299,Y -66.204,Z 81,A -121.7211,B 24.9111,C -2.1765,E1 24.9287,E2 206.2379} C_DIS
LIN {X -34.7225,Y -64.9658,Z 81,A -123.8585,B 24.911,C -2.1787,E1 24.9234,E2 208.376} C_DIS
LIN {X -37.1093,Y -63.6324,Z 81,A -126.0146,B 24.9108,C -2.1809,E1 24.9181,E2 210.5332} C_DIS
LIN {X -39.7481,Y -62.0169,Z 81,A -128.3314,B 24.9103,C -2.1867,E1 24.9127,E2 212.8434} C_DIS
LIN {X -42.0943,Y -60.449,Z 81,A -130.4857,B 24.9099,C -2.1912,E1 24.9077,E2 214.9943} C_DIS
LIN {X -44.3212,Y -58.8358,Z 81,A -132.7461,B 24.9099,C -2.1919,E1 24.9026,E2 217.261} C_DIS
LIN {X -46.7408,Y -56.9342,Z 81,A -135.2313,B 24.9097,C -2.1941,E1 24.8972,E2 219.7504} C_DIS
LIN {X -49.1253,Y -54.8881,Z 81,A -137.634,B 24.9092,C -2.1998,E1 24.8921,E2 222.149} C_DIS
LIN {X -51.4472,Y -52.7199,Z 81,A -140.1629,B 24.9089,C -2.2034,E1 24.887,E2 224.6796} C_DIS
LIN {X -53.49,Y -50.6447,Z 81,A -142.4113,B 24.9085,C -2.2086,E1 24.8827,E2 226.9253} C_DIS
LIN {X -55.6273,Y -48.2872,Z 81,A -144.9179,B 24.9081,C -2.2134,E1 24.878,E2 229.4318} C_DIS
LIN {X -57.6733,Y -45.8239,Z 81,A -147.3503,B 24.9075,C -2.2206,E1 24.8738,E2 231.8584} C_DIS
LIN {X -59.4069,Y -43.5525,Z 81,A -149.5252,B 24.907,C -2.227,E1 24.8701,E2 234.0283} C_DIS
LIN {X -60.9654,Y -41.3428,Z 81,A -151.6391,B 24.9065,C -2.232,E1 24.8668,E2 236.1407} C_DIS
LIN {X -62.442,Y -39.0769,Z 81,A -153.7556,B 24.9061,C -2.2371,E1 24.8636,E2 238.2558} C_DIS
LIN {X -63.8934,Y -36.6557,Z 81,A -155.9194,B 24.9056,C -2.2436,E1 24.8605,E2 240.4152} C_DIS
LIN {X -65.4835,Y -33.7339,Z 81,A -158.6953,B 24.9053,C -2.2462,E1 24.8569,E2 243.1996} C_DIS
LIN {X -66.8131,Y -31.0164,Z 81,A -161.0885,B 24.9049,C -2.2518,E1 24.854,E2 245.5924} C_DIS
LIN {X -68.0584,Y -28.1826,Z 81,A -163.4609,B 24.9042,C -2.2595,E1 24.8514,E2 247.9598} C_DIS
LIN {X -69.1813,Y -25.2973,Z 81,A -165.8512,B 24.9036,C -2.2669,E1 24.849,E2 250.3459} C_DIS
LIN {X -70.0768,Y -22.699,Z 81,A -167.9365,B 24.903,C -2.2744,E1 24.8472,E2 252.4252} C_DIS
LIN {X -70.8923,Y -20.0074,Z 81,A -170.2888,B 24.9027,C -2.2771,E1 24.8454,E2 254.7845} C_DIS
LIN {X -71.6699,Y -17.0186,Z 81,A -172.7149,B 24.9021,C -2.2839,E1 24.8437,E2 257.2087} C_DIS
LIN {X -72.3556,Y -13.809,Z 81,A -175.2762,B 24.9015,C -2.2915,E1 24.8423,E2 259.7667} C_DIS
LIN {X -72.8693,Y -10.782,Z 81,A -177.6265,B 24.9008,C -2.2998,E1 24.8413,E2 262.1114} C_DIS
LIN {X -73.2505,Y -7.7705,Z 81,A -179.9277,B 24.9,C -2.3085,E1 24.8405,E2 264.4054} C_DIS
LIN {X -73.5087,Y -4.7462,Z 81,A 177.5826,B 24.8996,C -2.3131,E1 24.84,E2 266.8993} C_DIS
LIN {X -73.6409,Y -1.7911,Z 81,A 175.242,B 24.8991,C -2.3194,E1 24.8398,E2 269.2387} C_DIS
LIN {X -73.6518,Y 1.2004,Z 81,A 173.0087,B 24.8982,C -2.3289,E1 24.8398,E2 271.4628} C_DIS
LIN {X -73.5529,Y 3.9971,Z 81,A 170.8177,B 24.8977,C -2.3355,E1 24.8401,E2 273.6511} C_DIS
LIN {X -73.3399,Y 6.876,Z 81,A 168.6394,B 24.8969,C -2.3442,E1 24.8406,E2 275.8219} C_DIS
LIN {X -73.055,Y 9.4329,Z 81,A 166.5815,B 24.8964,C -2.3493,E1 24.8413,E2 277.88} C_DIS
LIN {X -72.6414,Y 12.2161,Z 81,A 164.2263,B 24.8962,C -2.3525,E1 24.8423,E2 280.2416} C_DIS
LIN {X -72.0669,Y 15.2503,Z 81,A 161.8567,B 24.8954,C -2.3607,E1 24.8436,E2 282.6054} C_DIS
LIN {X -71.4531,Y 17.9069,Z 81,A 159.7211,B 24.8949,C -2.3671,E1 24.845,E2 284.7384} C_DIS
LIN {X -70.7487,Y 20.5142,Z 81,A 157.6364,B 24.8942,C -2.374,E1 24.8466,E2 286.8187} C_DIS
LIN {X -69.9425,Y 23.1138,Z 81,A 155.473,B 24.8938,C -2.3794,E1 24.8484,E2 288.9814} C_DIS
LIN {X -69.0472,Y 25.6651,Z 81,A 153.3925,B 24.8931,C -2.3864,E1 24.8504,E2 291.0572} C_DIS
LIN {X -68.0587,Y 28.1818,Z 81,A 151.2376,B 24.8927,C -2.3915,E1 24.8527,E2 293.2117} C_DIS
LIN {X -66.814,Y 31.0146,Z 81,A 148.912,B 24.8919,C -2.4006,E1 24.8553,E2 295.5285} C_DIS
LIN {X -65.6195,Y 33.4677,Z 81,A 146.7701,B 24.8913,C -2.4063,E1 24.858,E2 297.6681} C_DIS
LIN {X -64.3368,Y 35.8718,Z 81,A 144.646,B 24.8908,C -2.4124,E1 24.8608,E2 299.7891} C_DIS
LIN {X -62.9143,Y 38.3119,Z 81,A 142.2829,B 24.8906,C -2.4148,E1 24.8642,E2 302.1586} C_DIS
LIN {X -61.2487,Y 40.9244,Z 81,A 139.9067,B 24.8899,C -2.4222,E1 24.8678,E2 304.5291} C_DIS
LIN {X -59.6887,Y 43.1677,Z 81,A 137.774,B 24.8894,C -2.4278,E1 24.8713,E2 306.6589} C_DIS
LIN {X -57.9437,Y 45.4818,Z 81,A 135.5125,B 24.8889,C -2.4336,E1 24.8751,E2 308.9173} C_DIS
LIN {X -55.9427,Y 47.9214,Z 81,A 133.0031,B 24.8884,C -2.4386,E1 24.8796,E2 311.4263} C_DIS
LIN {X -53.8192,Y 50.2946,Z 81,A 130.552,B 24.8878,C -2.4453,E1 24.8842,E2 313.8721} C_DIS
LIN {X -51.6175,Y 52.5518,Z 81,A 128.0455,B 24.8873,C -2.4499,E1 24.8891,E2 316.3782} C_DIS
LIN {X -49.3199,Y 54.714,Z 81,A 125.6206,B 24.8868,C -2.4562,E1 24.8941,E2 318.798} C_DIS
LIN {X -46.8859,Y 56.8135,Z 81,A 123.0746,B 24.8864,C -2.4607,E1 24.8995,E2 321.3431} C_DIS
LIN {X -44.5945,Y 58.6305,Z 81,A 120.8511,B 24.8858,C -2.4666,E1 24.9044,E2 323.5606} C_DIS
LIN {X -42.4112,Y 60.2287,Z 81,A 118.7356,B 24.8854,C -2.4706,E1 24.9092,E2 325.674} C_DIS
LIN {X -40.1705,Y 61.7457,Z 81,A 116.6205,B 24.8851,C -2.4744,E1 24.9141,E2 327.787} C_DIS
LIN {X -37.8756,Y 63.1795,Z 81,A 114.4693,B 24.8848,C -2.4771,E1 24.9193,E2 329.9384} C_DIS
LIN {X -35.3669,Y 64.6163,Z 81,A 112.2077,B 24.8845,C -2.4807,E1 24.9248,E2 332.198} C_DIS
LIN {X -32.6278,Y 66.0412,Z 81,A 109.8783,B 24.884,C -2.4863,E1 24.9306,E2 334.5204} C_DIS
LIN {X -30.2963,Y 67.1427,Z 81,A 107.8902,B 24.8836,C -2.4898,E1 24.9356,E2 336.5052} C_DIS
LIN {X -27.8153,Y 68.2079,Z 81,A 105.7851,B 24.8834,C -2.4926,E1 24.941,E2 338.6083} C_DIS
LIN {X -25.2956,Y 69.1819,Z 81,A 103.6563,B 24.8832,C -2.4947,E1 24.9466,E2 340.7366} C_DIS
LIN {X -22.7109,Y 70.073,Z 81,A 101.5457,B 24.8829,C -2.4976,E1 24.9521,E2 342.8443} C_DIS
LIN {X -19.9228,Y 70.9162,Z 81,A 99.129,B 24.883,C -2.4963,E1 24.9586,E2 345.2679} C_DIS
LIN {X -16.9801,Y 71.6788,Z 81,A 96.8522,B 24.8826,C -2.5007,E1 24.9648,E2 347.5375} C_DIS
LIN {X -14.3612,Y 72.2493,Z 81,A 94.7172,B 24.8826,C -2.5012,E1 24.9706,E2 349.6738} C_DIS
LIN {X -11.7205,Y 72.7243,Z 81,A 92.6094,B 24.8825,C -2.5022,E1 24.9764,E2 351.7813} C_DIS
LIN {X -8.6224,Y 73.1551,Z 81,A 90.2878,B 24.8821,C -2.5065,E1 24.9828,E2 354.0944} C_DIS
LIN {X -5.8099,Y 73.432,Z 81,A 88.0516,B 24.8821,C -2.5065,E1 24.9891,E2 356.3315} C_DIS
LIN {X -3.2099,Y 73.5915,Z 81,A 86.058,B 24.8819,C -2.5081,E1 24.9946,E2 358.322} C_DIS
LIN {X -0.5043,Y 73.6597,Z 81,A 83.9526,B 24.8819,C -2.5086,E1 25.0005,E2 360.4263} C_DIS
LIN {X 2.3207,Y 73.6249,Z 81,A 81.6575,B 24.8821,C -2.5064,E1 25.0069,E2 362.7262} C_DIS
LIN {X 5.5263,Y 73.4546,Z 81,A 79.1986,B 24.882,C -2.5074,E1 25.0138,E2 365.1818} C_DIS
LIN {X 8.146,Y 73.2108,Z 81,A 77.0993,B 24.8821,C -2.5057,E1 25.0196,E2 367.2837} C_DIS
LIN {X 11.3038,Y 72.789,Z 81,A 74.7351,B 24.8819,C -2.5081,E1 25.0261,E2 369.6402} C_DIS
LIN {X 13.9159,Y 72.335,Z 81,A 72.6765,B 24.8819,C -2.5074,E1 25.0318,E2 371.6982} C_DIS
LIN {X 16.648,Y 71.7555,Z 81,A 70.5245,B 24.882,C -2.5068,E1 25.0376,E2 373.8486} C_DIS
LIN {X 19.2992,Y 71.0884,Z 81,A 68.4233,B 24.882,C -2.5062,E1 25.0433,E2 375.948} C_DIS
LIN {X 21.7768,Y 70.3689,Z 81,A 66.376,B 24.8823,C -2.5037,E1 25.0488,E2 377.9978} C_DIS
LIN {X 24.4532,Y 69.4842,Z 81,A 64.2367,B 24.8823,C -2.5033,E1 25.0544,E2 380.1339} C_DIS
LIN {X 26.8747,Y 68.584,Z 81,A 62.1828,B 24.8827,C -2.5002,E1 25.0598,E2 382.1907} C_DIS
LIN {X 29.4797,Y 67.5052,Z 81,A 59.838,B 24.8833,C -2.4938,E1 25.0658,E2 384.5451} C_DIS
LIN {X 32.3131,Y 66.1972,Z 81,A 57.4985,B 24.8833,C -2.4933,E1 25.0717,E2 386.8797} C_DIS
LIN {X 34.747,Y 64.9526,Z 81,A 55.3956,B 24.8835,C -2.4911,E1 25.0769,E2 388.9818} C_DIS
LIN {X 37.1037,Y 63.6358,Z 81,A 53.2613,B 24.8839,C -2.4872,E1 25.0821,E2 391.119} C_DIS
LIN {X 39.741,Y 62.0214,Z 81,A 50.9636,B 24.8839,C -2.4866,E1 25.0875,E2 393.4109} C_DIS
LIN {X 42.0247,Y 60.4974,Z 81,A 48.7592,B 24.8844,C -2.4812,E1 25.0926,E2 395.6206} C_DIS
LIN {X 44.6495,Y 58.5882,Z 81,A 46.2107,B 24.8849,C -2.4761,E1 25.0984,E2 398.1719} C_DIS
LIN {X 47.0864,Y 56.6469,Z 81,A 43.7914,B 24.8853,C -2.4718,E1 25.1036,E2 400.5924} C_DIS
LIN {X 49.4727,Y 54.577,Z 81,A 41.3069,B 24.8858,C -2.4662,E1 25.1088,E2 403.0802} C_DIS
LIN {X 51.7655,Y 52.4055,Z 81,A 38.9008,B 24.8862,C -2.4626,E1 25.1136,E2 405.4849} C_DIS
LIN {X 53.9649,Y 50.1397,Z 81,A 36.4161,B 24.8868,C -2.4564,E1 25.1184,E2 407.9734} C_DIS
LIN {X 56.064,Y 47.779,Z 81,A 33.9902,B 24.8872,C -2.4517,E1 25.1229,E2 410.3994} C_DIS
LIN {X 58.0882,Y 45.2984,Z 81,A 31.5908,B 24.8875,C -2.4484,E1 25.127,E2 412.7954} C_DIS
LIN {X 59.7073,Y 43.142,Z 81,A 29.4466,B 24.8881,C -2.442,E1 25.1306,E2 414.9445} C_DIS
LIN {X 61.4624,Y 40.6003,Z 81,A 27.172,B 24.8883,C -2.4396,E1 25.1342,E2 417.2135} C_DIS
LIN {X 62.9077,Y 38.3227,Z 81,A 25.0765,B 24.8888,C -2.4342,E1 25.1372,E2 419.3111} C_DIS
LIN {X 64.3424,Y 35.8617,Z 81,A 22.931,B 24.8891,C -2.4304,E1 25.1402,E2 421.4546} C_DIS
LIN {X 65.6204,Y 33.4659,Z 81,A 20.8079,B 24.8897,C -2.4243,E1 25.143,E2 423.5809} C_DIS
LIN {X 66.8178,Y 31.0064,Z 81,A 18.5207,B 24.8907,C -2.4138,E1 25.1457,E2 425.8806} C_DIS
LIN {X 68.0577,Y 28.1843,Z 81,A 16.1507,B 24.8912,C -2.4077,E1 25.1483,E2 428.2518} C_DIS
LIN {X 69.1766,Y 25.3103,Z 81,A 13.9003,B 24.8914,C -2.4051,E1 25.1505,E2 430.496} C_DIS
LIN {X 70.0549,Y 22.7668,Z 81,A 11.8079,B 24.892,C -2.3989,E1 25.1524,E2 432.5911} C_DIS
LIN {X 70.8863,Y 20.0284,Z 81,A 9.4595,B 24.8929,C -2.3887,E1 25.1543,E2 434.9502} C_DIS
LIN {X 71.6704,Y 17.0163,Z 81,A 7.1437,B 24.8933,C -2.3844,E1 25.1558,E2 437.2628} C_DIS
LIN {X 72.2474,Y 14.3709,Z 81,A 5.0127,B 24.894,C -2.3772,E1 25.157,E2 439.3984} C_DIS
LIN {X 72.7267,Y 11.706,Z 81,A 2.9219,B 24.8945,C -2.3711,E1 25.158,E2 441.4913} C_DIS
LIN {X 73.156,Y 8.6139,Z 81,A 0.5821,B 24.8949,C -2.3661,E1 25.1588,E2 443.8292} C_DIS
LIN {X 73.4324,Y 5.8046,Z 81,A -1.5199,B 24.8953,C -2.362,E1 25.1594,E2 445.9286} C_DIS
LIN {X 73.5909,Y 3.2228,Z 81,A -3.566,B 24.896,C -2.3546,E1 25.1597,E2 447.9798} C_DIS
LIN {X 73.6571,Y 0.9103,Z 81,A -5.4152,B 24.8966,C -2.3474,E1 25.1597,E2 449.835} C_DIS
LIN {X 73.6404,Y -1.8156,Z 81,A -7.5587,B 24.8973,C -2.34,E1 25.1597,E2 451.9833} C_DIS
LIN {X 73.4976,Y -4.9104,Z 81,A -9.8505,B 24.8976,C -2.3358,E1 25.1593,E2 454.2714} C_DIS
LIN {X 73.2676,Y -7.6069,Z 81,A -11.9422,B 24.8982,C -2.3294,E1 25.1588,E2 456.3657} C_DIS
LIN {X 72.9388,Y -10.2929,Z 81,A -14.0337,B 24.8987,C -2.3231,E1 25.158,E2 458.4597} C_DIS
LIN {X 72.4652,Y -13.2228,Z 81,A -16.2368,B 24.8991,C -2.3189,E1 25.157,E2 460.66} C_DIS
LIN {X 71.9561,Y -15.7583,Z 81,A -18.4716,B 24.9002,C -2.306,E1 25.1557,E2 462.9122} C_DIS
LIN {X 71.2311,Y -18.7707,Z 81,A -20.8548,B 24.9008,C -2.2992,E1 25.1541,E2 465.2977} C_DIS
LIN {X 70.3405,Y -21.8684,Z 81,A -23.1974,B 24.9011,C -2.2962,E1 25.1522,E2 467.6339} C_DIS
LIN {X 69.4776,Y -24.472,Z 81,A -25.402,B 24.9018,C -2.2876,E1 25.1502,E2 469.8466} C_DIS
LIN {X 68.3915,Y -27.3642,Z 81,A -27.7716,B 24.9024,C -2.2812,E1 25.1478,E2 472.218} C_DIS
LIN {X 67.3404,Y -29.8576,Z 81,A -29.8637,B 24.9029,C -2.2752,E1 25.1455,E2 474.3128} C_DIS
LIN {X 66.1983,Y -32.311,Z 81,A -31.9562,B 24.9034,C -2.2694,E1 25.143,E2 476.4079} C_DIS
LIN {X 64.9465,Y -34.7581,Z 81,A -34.0705,B 24.9039,C -2.2638,E1 25.1403,E2 478.5241} C_DIS
LIN {X 63.6312,Y -37.1114,Z 81,A -36.1957,B 24.9044,C -2.2569,E1 25.1373,E2 480.6546} C_DIS
LIN {X 62.0178,Y -39.7467,Z 81,A -38.4869,B 24.9047,C -2.2534,E1 25.1339,E2 482.9424} C_DIS
LIN {X 60.4075,Y -42.154,Z 81,A -40.7383,B 24.9053,C -2.2473,E1 25.1304,E2 485.1973} C_DIS
LIN {X 58.8,Y -44.3688,Z 81,A -42.9064,B 24.9058,C -2.2404,E1 25.1268,E2 487.3712} C_DIS
LIN {X 56.9173,Y -46.7611,Z 81,A -45.3223,B 24.9065,C -2.2328,E1 25.1225,E2 489.7939} C_DIS
LIN {X 54.8798,Y -49.1347,Z 81,A -47.7077,B 24.9069,C -2.228,E1 25.1181,E2 492.1798} C_DIS
LIN {X 52.8102,Y -51.3536,Z 81,A -50.0916,B 24.9074,C -2.2215,E1 25.1135,E2 494.5688} C_DIS
LIN {X 50.613,Y -53.5198,Z 81,A -52.4386,B 24.9078,C -2.2173,E1 25.1088,E2 496.9158} C_DIS
LIN {X 48.2957,Y -55.6199,Z 81,A -54.901,B 24.9083,C -2.2109,E1 25.1037,E2 499.3836} C_DIS
LIN {X 45.7969,Y -57.6946,Z 81,A -57.3504,B 24.9086,C -2.2076,E1 25.0984,E2 501.8316} C_DIS
LIN {X 43.5432,Y -59.4137,Z 81,A -59.4825,B 24.9088,C -2.205,E1 25.0936,E2 503.962} C_DIS
LIN {X 41.3376,Y -60.9689,Z 81,A -61.5705,B 24.9091,C -2.2012,E1 25.0888,E2 506.0522} C_DIS
LIN {X 39.075,Y -62.4432,Z 81,A -63.662,B 24.9094,C -2.1974,E1 25.0839,E2 508.1458} C_DIS
LIN {X 36.6573,Y -63.8925,Z 81,A -65.8109,B 24.9097,C -2.1947,E1 25.0787,E2 510.2946} C_DIS
LIN {X 34.2639,Y -65.2073,Z 81,A -67.9162,B 24.9099,C -2.1915,E1 25.0735,E2 512.4012} C_DIS
LIN {X 31.9523,Y -66.3706,Z 81,A -69.9514,B 24.9102,C -2.1877,E1 25.0684,E2 514.4401} C_DIS
LIN {X 29.3566,Y -67.5589,Z 81,A -72.1802,B 24.9105,C -2.1841,E1 25.0627,E2 516.6719} C_DIS
LIN {X 26.8182,Y -68.6061,Z 81,A -74.4563,B 24.9111,C -2.1772,E1 25.0568,E2 518.9591} C_DIS
LIN {X 23.9484,Y -69.6611,Z 81,A -76.8356,B 24.9113,C -2.1742,E1 25.0505,E2 521.3408} C_DIS
LIN {X 21.0277,Y -70.5964,Z 81,A -79.065,B 24.9113,C -2.1757,E1 25.0446,E2 523.5626} C_DIS
LIN {X 18.4559,Y -71.312,Z 81,A -81.166,B 24.9114,C -2.1728,E1 25.0389,E2 525.667} C_DIS
LIN {X 15.753,Y -71.9573,Z 81,A -83.2903,B 24.9115,C -2.1718,E1 25.0332,E2 527.7909} C_DIS
LIN {X 12.9819,Y -72.5085,Z 81,A -85.4371,B 24.9115,C -2.1714,E1 25.0273,E2 529.9362} C_DIS
LIN {X 10.2883,Y -72.9394,Z 81,A -87.7551,B 24.9121,C -2.1646,E1 25.0208,E2 532.268} C_DIS
LIN {X 7.2123,Y -73.3088,Z 81,A -90.1114,B 24.9121,C -2.1646,E1 25.0143,E2 534.6227} C_DIS
LIN {X 4.514,Y -73.5243,Z 81,A -92.1776,B 24.9121,C -2.1647,E1 25.0085,E2 536.6877} C_DIS
LIN {X 1.6361,Y -73.6438,Z 81,A -94.465,B 24.9123,C -2.1628,E1 25.0022,E2 538.9793} C_DIS
LIN {X 1.6361,Y -73.6438,Z 81,A -94.465,B 24.9123,C -2.1628,E1 25.0022,E2 538.9793} C_DIS
Enddeposition()
LIN {X 0.5451,Y -82.9088,Z 82,A -94.4611,B 24.9226,C -2.0321,E1 25.0013,E2 539.2853} C_DIS
Startdeposition()
$VEL.CP = VEL_PRINT
LIN {X 3.0518,Y -82.856,Z 82,A -92.3384,B 24.9216,C -2.0445,E1 25.0073,E2 537.1337} C_DIS
LIN {X 5.2143,Y -82.7474,Z 82,A -90.9675,B 24.9219,C -2.0413,E1 25.0111,E2 535.7709} C_DIS
LIN {X 7.1801,Y -82.6003,Z 82,A -89.4638,B 24.9215,C -2.0463,E1 25.0153,E2 534.2561} C_DIS
LIN {X 9.1388,Y -82.407,Z 82,A -88.1646,B 24.9215,C -2.0452,E1 25.0189,E2 532.9604} C_DIS
LIN {X 11.3636,Y -82.1287,Z 82,A -86.7505,B 24.9218,C -2.042,E1 25.0228,E2 531.555} C_DIS
LIN {X 13.2371,Y -81.8483,Z 82,A -85.3529,B 24.9215,C -2.0457,E1 25.0267,E2 530.15} C_DIS
LIN {X 15.2418,Y -81.4988,Z 82,A -83.9061,B 24.9213,C -2.0481,E1 25.0307,E2 528.6992} C_DIS
LIN {X 17.2373,Y -81.1002,Z 82,A -82.5025,B 24.9213,C -2.0492,E1 25.0345,E2 527.2947} C_DIS
LIN {X 19.1575,Y -80.6686,Z 82,A -81.1456,B 24.9212,C -2.0504,E1 25.0382,E2 525.9369} C_DIS
LIN {X 21.1959,Y -80.1567,Z 82,A -79.6961,B 24.9211,C -2.0518,E1 25.0421,E2 524.4862} C_DIS
LIN {X 23.7078,Y -79.4489,Z 82,A -77.7942,B 24.9207,C -2.0569,E1 25.0473,E2 522.5755} C_DIS
LIN {X 26.008,Y -78.7274,Z 82,A -76.2359,B 24.9207,C -2.0555,E1 25.0514,E2 521.0234} C_DIS
LIN {X 27.995,Y -78.0426,Z 82,A -74.8305,B 24.9207,C -2.0559,E1 25.0551,E2 519.6199} C_DIS
LIN {X 29.9018,Y -77.3321,Z 82,A -73.3853,B 24.9205,C -2.059,E1 25.0589,E2 518.1705} C_DIS
LIN {X 31.7906,Y -76.5749,Z 82,A -72.0265,B 24.9205,C -2.0595,E1 25.0624,E2 516.8136} C_DIS
LIN {X 33.5994,Y -75.7991,Z 82,A -70.4393,B 24.9197,C -2.0687,E1 25.0665,E2 515.2084} C_DIS
LIN {X 36.3666,Y -74.5111,Z 82,A -68.5257,B 24.92,C -2.0658,E1 25.0713,E2 513.3066} C_DIS
LIN {X 38.2619,Y -73.5552,Z 82,A -67.1208,B 24.92,C -2.0663,E1 25.0748,E2 511.9045} C_DIS
LIN {X 40.0372,Y -72.6043,Z 82,A -65.6777,B 24.9196,C -2.0703,E1 25.0783,E2 510.456} C_DIS
LIN {X 41.8069,Y -71.5999,Z 82,A -64.0463,B 24.9189,C -2.0801,E1 25.0823,E2 508.8064} C_DIS
LIN {X 44.56,Y -69.9189,Z 82,A -62.1277,B 24.9193,C -2.0743,E1 25.0868,E2 506.9076} C_DIS
LIN {X 46.9609,Y -68.3304,Z 82,A -60.119,B 24.919,C -2.0788,E1 25.0915,E2 504.895} C_DIS
LIN {X 48.5698,Y -67.1968,Z 82,A -58.6821,B 24.9185,C -2.0841,E1 25.0948,E2 503.4507} C_DIS
LIN {X 50.2571,Y -65.9438,Z 82,A -57.2765,B 24.9185,C -2.0856,E1 25.0979,E2 502.0465} C_DIS
LIN {X 51.8603,Y -64.6906,Z 82,A -55.6725,B 24.9177,C -2.0951,E1 25.1014,E2 500.4261} C_DIS
LIN {X 54.2063,Y -62.7379,Z 82,A -53.8208,B 24.918,C -2.0914,E1 25.1053,E2 498.5903} C_DIS
LIN {X 55.6804,Y -61.4339,Z 82,A -52.3848,B 24.9175,C -2.097,E1 25.1083,E2 497.1467} C_DIS
LIN {X 57.2194,Y -60.0026,Z 82,A -50.98,B 24.9174,C -2.0989,E1 25.1112,E2 495.7433} C_DIS
LIN {X 58.6278,Y -58.6278,Z 82,A -49.6272,B 24.9171,C -2.1019,E1 25.1139,E2 494.389} C_DIS
LIN {X 60.0489,Y -57.1713,Z 82,A -48.1161,B 24.9166,C -2.1088,E1 25.1168,E2 492.8682} C_DIS
LIN {X 62.1125,Y -54.9223,Z 82,A -46.0907,B 24.9164,C -2.1114,E1 25.1206,E2 490.8458} C_DIS
LIN {X 63.4417,Y -53.3815,Z 82,A -44.7326,B 24.9162,C -2.1134,E1 25.1231,E2 489.489} C_DIS
LIN {X 64.7326,Y -51.8085,Z 82,A -43.2453,B 24.9157,C -2.1198,E1 25.1257,E2 487.9936} C_DIS
LIN {X 65.9846,Y -50.2042,Z 82,A -41.8963,B 24.9156,C -2.1216,E1 25.128,E2 486.6465} C_DIS
LIN {X 67.5726,Y -48.0431,Z 82,A -39.993,B 24.915,C -2.1283,E1 25.1311,E2 484.7366} C_DIS
LIN {X 68.9757,Y -46.0078,Z 82,A -38.4388,B 24.915,C -2.128,E1 25.1335,E2 483.191} C_DIS
LIN {X 70.084,Y -44.3012,Z 82,A -37.0412,B 24.9148,C -2.1316,E1 25.1356,E2 481.7918} C_DIS
LIN {X 71.1161,Y -42.6254,Z 82,A -35.6472,B 24.9144,C -2.1366,E1 25.1377,E2 480.3931} C_DIS
LIN {X 72.1408,Y -40.8673,Z 82,A -34.2097,B 24.914,C -2.1417,E1 25.1397,E2 478.951} C_DIS
LIN {X 73.1531,Y -39.0255,Z 82,A -32.714,B 24.9135,C -2.1474,E1 25.1417,E2 477.4498} C_DIS
LIN {X 74.0888,Y -37.2185,Z 82,A -31.4522,B 24.9135,C -2.1467,E1 25.1433,E2 476.1963} C_DIS
LIN {X 74.9517,Y -35.4495,Z 82,A -30.018,B 24.913,C -2.1532,E1 25.145,E2 474.7545} C_DIS
LIN {X 75.8258,Y -33.5382,Z 82,A -28.6251,B 24.9128,C -2.1556,E1 25.1466,E2 473.3634} C_DIS
LIN {X 76.6009,Y -31.7291,Z 82,A -27.2644,B 24.9125,C -2.1597,E1 25.1481,E2 472.0005} C_DIS
LIN {X 77.3801,Y -29.7773,Z 82,A -25.5882,B 24.9115,C -2.1716,E1 25.1498,E2 470.3054} C_DIS
LIN {X 78.4237,Y -26.9089,Z 82,A -23.7693,B 24.9118,C -2.1684,E1 25.1515,E2 468.5042} C_DIS
LIN {X 79.0407,Y -25.04,Z 82,A -22.3357,B 24.9113,C -2.1751,E1 25.1527,E2 467.063} C_DIS
LIN {X 79.6314,Y -23.0927,Z 82,A -20.979,B 24.911,C -2.1779,E1 25.1538,E2 465.7077} C_DIS
LIN {X 80.1907,Y -21.0668,Z 82,A -19.537,B 24.9107,C -2.1821,E1 25.1548,E2 464.264} C_DIS
LIN {X 80.6686,Y -19.1575,Z 82,A -18.1861,B 24.9104,C -2.186,E1 25.1557,E2 462.9116} C_DIS
LIN {X 81.1144,Y -17.1721,Z 82,A -16.7896,B 24.91,C -2.1902,E1 25.1565,E2 461.5134} C_DIS
LIN {X 81.5232,Y -15.1105,Z 82,A -15.2531,B 24.9094,C -2.1976,E1 25.1574,E2 459.9684} C_DIS
LIN {X 81.8695,Y -13.1053,Z 82,A -13.9937,B 24.9094,C -2.1972,E1 25.1579,E2 458.7173} C_DIS
LIN {X 82.1665,Y -11.0922,Z 82,A -12.5546,B 24.909,C -2.2028,E1 25.1585,E2 457.2736} C_DIS
LIN {X 82.5129,Y -8.1268,Z 82,A -10.466,B 24.9084,C -2.2102,E1 25.1591,E2 455.1797} C_DIS
LIN {X 82.6875,Y -6.0994,Z 82,A -9.1099,B 24.9081,C -2.213,E1 25.1594,E2 453.825} C_DIS
LIN {X 82.8152,Y -4.0016,Z 82,A -7.7101,B 24.9079,C -2.2159,E1 25.1596,E2 452.4267} C_DIS
LIN {X 82.8884,Y -1.968,Z 82,A -6.3137,B 24.9075,C -2.2201,E1 25.1598,E2 451.0287} C_DIS
LIN {X 82.9089,Y 0.6054,Z 82,A -4.2996,B 24.9064,C -2.2336,E1 25.1598,E2 448.9946} C_DIS
LIN {X 82.856,Y 3.0518,Z 82,A -2.786,B 24.9064,C -2.2331,E1 25.1596,E2 447.4914} C_DIS
LIN {X 82.7516,Y 5.1508,Z 82,A -1.4262,B 24.9064,C -2.2346,E1 25.1594,E2 446.1361} C_DIS
LIN {X 82.6003,Y 7.1801,Z 82,A 0.0148,B 24.9059,C -2.2402,E1 25.1591,E2 444.6903} C_DIS
LIN {X 82.3992,Y 9.2051,Z 82,A 1.3665,B 24.9056,C -2.2428,E1 25.1587,E2 443.3405} C_DIS
LIN {X 82.1485,Y 11.2245,Z 82,A 2.763,B 24.9053,C -2.2469,E1 25.1582,E2 441.9426} C_DIS
LIN {X 81.8483,Y 13.2371,Z 82,A 4.1598,B 24.9049,C -2.251,E1 25.1576,E2 440.5444} C_DIS
LIN {X 81.4988,Y 15.2418,Z 82,A 5.5992,B 24.9045,C -2.2565,E1 25.1569,E2 439.1005} C_DIS
LIN {X 80.8826,Y 18.2312,Z 82,A 7.6511,B 24.9041,C -2.261,E1 25.1557,E2 437.0497} C_DIS
LIN {X 80.4236,Y 20.1609,Z 82,A 9.0864,B 24.9036,C -2.2674,E1 25.1547,E2 435.6078} C_DIS
LIN {X 79.9088,Y 22.1137,Z 82,A 10.4418,B 24.9033,C -2.2702,E1 25.1537,E2 434.2534} C_DIS
LIN {X 79.3222,Y 24.1319,Z 82,A 12.1145,B 24.9023,C -2.2819,E1 25.1524,E2 432.5627} C_DIS
LIN {X 78.4024,Y 26.9722,Z 82,A 13.9748,B 24.9023,C -2.2813,E1 25.1508,E2 430.7144} C_DIS
LIN {X 77.7168,Y 28.8881,Z 82,A 15.3319,B 24.9021,C -2.2838,E1 25.1495,E2 429.3589} C_DIS
LIN {X 76.9593,Y 30.8485,Z 82,A 16.7749,B 24.9018,C -2.2877,E1 25.148,E2 427.9148} C_DIS
LIN {X 76.1791,Y 32.7279,Z 82,A 18.2133,B 24.9014,C -2.2927,E1 25.1464,E2 426.4723} C_DIS
LIN {X 75.1618,Y 34.9982,Z 82,A 20.0222,B 24.9007,C -2.3006,E1 25.1443,E2 424.6547} C_DIS
LIN {X 74.0288,Y 37.3377,Z 82,A 21.7806,B 24.9004,C -2.3043,E1 25.1421,E2 422.897} C_DIS
LIN {X 72.4629,Y 40.2905,Z 82,A 24.129,B 24.8997,C -2.3118,E1 25.139,E2 420.543} C_DIS
LIN {X 70.5877,Y 43.4949,Z 82,A 26.5533,B 24.8995,C -2.3139,E1 25.1355,E2 418.1263} C_DIS
LIN {X 69.4623,Y 45.2698,Z 82,A 27.9573,B 24.8994,C -2.3161,E1 25.1334,E2 416.7242} C_DIS
LIN {X 68.3304,Y 46.9609,Z 82,A 29.3132,B 24.8992,C -2.318,E1 25.1313,E2 415.3705} C_DIS
LIN {X 67.1968,Y 48.5698,Z 82,A 30.7486,B 24.8987,C -2.3238,E1 25.1289,E2 413.9283} C_DIS
LIN {X 65.9438,Y 50.2571,Z 82,A 32.3311,B 24.898,C -2.3315,E1 25.1263,E2 412.3351} C_DIS
LIN {X 64.092,Y 52.5989,Z 82,A 34.3615,B 24.8977,C -2.3353,E1 25.1227,E2 410.3051} C_DIS
LIN {X 62.1528,Y 54.8762,Z 82,A 36.2646,B 24.8977,C -2.3347,E1 25.1192,E2 408.412} C_DIS
LIN {X 60.7002,Y 56.4787,Z 82,A 37.9855,B 24.8968,C -2.3453,E1 25.1159,E2 406.6736} C_DIS
LIN {X 58.6278,Y 58.6278,Z 82,A 39.8434,B 24.897,C -2.3431,E1 25.1123,E2 404.8288} C_DIS
LIN {X 57.1713,Y 60.0489,Z 82,A 41.2031,B 24.8969,C -2.3445,E1 25.1096,E2 403.4715} C_DIS
LIN {X 55.6307,Y 61.4784,Z 82,A 42.6491,B 24.8966,C -2.3472,E1 25.1066,E2 402.0249} C_DIS
LIN {X 54.1052,Y 62.8251,Z 82,A 44.0491,B 24.8964,C -2.3498,E1 25.1037,E2 400.6244} C_DIS
LIN {X 51.8085,Y 64.7326,Z 82,A 46.3123,B 24.8955,C -2.36,E1 25.0988,E2 398.3457} C_DIS
LIN {X 49.3369,Y 66.6351,Z 82,A 48.2082,B 24.8959,C -2.3556,E1 25.0946,E2 396.4671} C_DIS
LIN {X 47.7415,Y 67.7877,Z 82,A 49.6462,B 24.8955,C -2.3603,E1 25.0913,E2 395.0229} C_DIS
LIN {X 46.0078,Y 68.9757,Z 82,A 51.0534,B 24.8954,C -2.3612,E1 25.088,E2 393.6182} C_DIS
LIN {X 44.3578,Y 70.0486,Z 82,A 52.4085,B 24.8952,C -2.3632,E1 25.0848,E2 392.2629} C_DIS
LIN {X 42.6254,Y 71.1161,Z 82,A 53.8504,B 24.8949,C -2.3664,E1 25.0814,E2 390.8179} C_DIS
LIN {X 40.8673,Y 72.1408,Z 82,A 55.4438,B 24.8942,C -2.3742,E1 25.0775,E2 389.2107} C_DIS
LIN {X 38.1248,Y 73.6265,Z 82,A 57.3187,B 24.8947,C -2.3683,E1 25.0729,E2 387.3551} C_DIS
Enddeposition()
END
